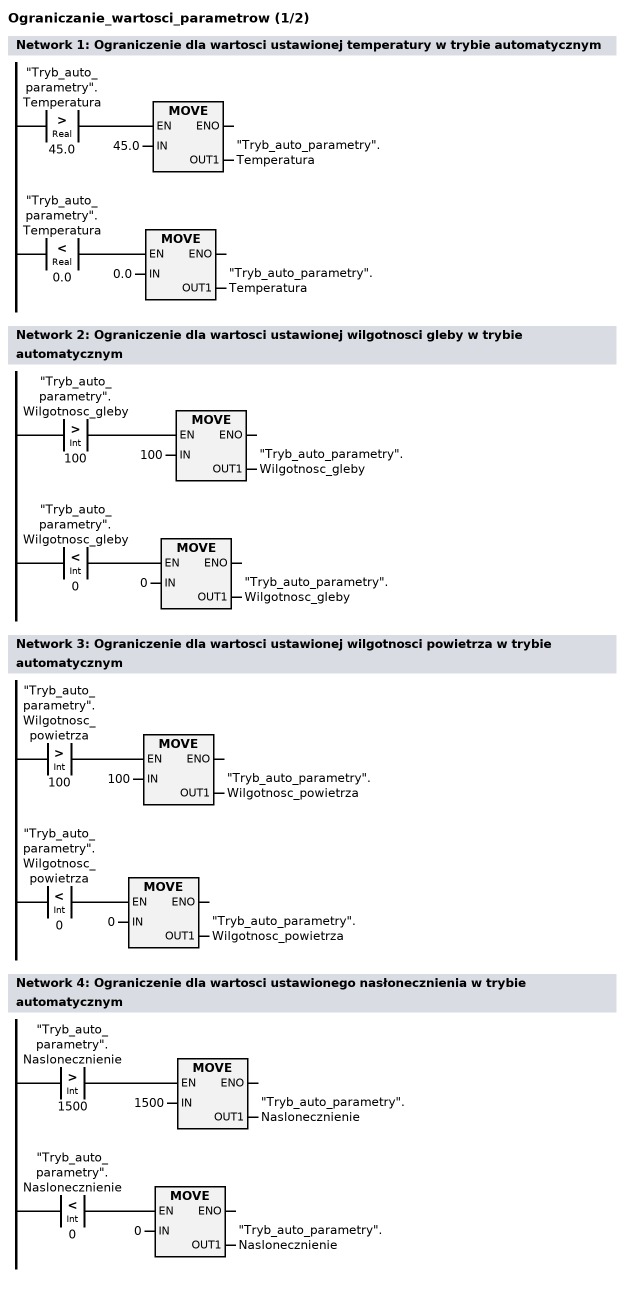
   RUNG wire#powerrail
      { S7_Templates := "SrcType := Real" } GT_Contact(in1 := "Tryb_auto_parametry".Temperatura, in2 := 45.0)
      Move(in := 45.0, out1 => "Tryb_auto_parametry".Temperatura)
   END_RUNG
   RUNG wire#powerrail
      { S7_Templates := "SrcType := Real" } LT_Contact(in1 := "Tryb_auto_parametry".Temperatura, in2 := 0.0)
      Move(in := 0.0, out1 => "Tryb_auto_parametry".Temperatura)
   END_RUNG
   // the same network as SCL:
   IF "Tryb_auto_parametry".Temperatura > 45.0 THEN "Tryb_auto_parametry".Temperatura := 45.0; END_IF;
   IF "Tryb_auto_parametry".Temperatura < 0.0 THEN "Tryb_auto_parametry".Temperatura := 0.0; END_IF;
END_REGION

REGION Network 2: Ograniczenie dla wartosci ustawionej wilgotnosci gleby w trybie automatycznym
   RUNG wire#powerrail
      { S7_Templates := "SrcType := Int" } GT_Contact(in1 := "Tryb_auto_parametry".Wilgotnosc_gleby, in2 := 100)
      Move(in := 100, out1 => "Tryb_auto_parametry".Wilgotnosc_gleby)
   END_RUNG
   RUNG wire#powerrail
      { S7_Templates := "SrcType := Int" } LT_Contact(in1 := "Tryb_auto_parametry".Wilgotnosc_gleby, in2 := 0)
      Move(in := 0, out1 => "Tryb_auto_parametry".Wilgotnosc_gleby)
   END_RUNG
   // the same network as SCL:
   IF "Tryb_auto_parametry".Wilgotnosc_gleby > 100 THEN
       "Tryb_auto_parametry".Wilgotnosc_gleby := 100;
   END_IF;
   IF "Tryb_auto_parametry".Wilgotnosc_gleby < 0 THEN "Tryb_auto_parametry".Wilgotnosc_gleby := 0; END_IF;
END_REGION

REGION Network 3: Ograniczenie dla wartosci ustawionej wilgotnosci powietrza w trybie automatycznym
   RUNG wire#powerrail
      { S7_Templates := "SrcType := Int" } GT_Contact(in1 := "Tryb_auto_parametry".Wilgotnosc_powietrza, in2 := 100)
      Move(in := 100, out1 => "Tryb_auto_parametry".Wilgotnosc_powietrza)
   END_RUNG
   RUNG wire#powerrail
      { S7_Templates := "SrcType := Int" } LT_Contact(in1 := "Tryb_auto_parametry".Wilgotnosc_powietrza, in2 := 0)
      Move(in := 0, out1 => "Tryb_auto_parametry".Wilgotnosc_powietrza)
   END_RUNG
   // the same network as SCL:
   IF "Tryb_auto_parametry".Wilgotnosc_powietrza > 100 THEN
       "Tryb_auto_parametry".Wilgotnosc_powietrza := 100;
   END_IF;
   IF "Tryb_auto_parametry".Wilgotnosc_powietrza < 0 THEN
       "Tryb_auto_parametry".Wilgotnosc_powietrza := 0;
   END_IF;
END_REGION

REGION Network 4: Ograniczenie dla wartosci ustawionego nasłonecznienia w trybie automatycznym
   RUNG wire#powerrail
      { S7_Templates := "SrcType := Int" } GT_Contact(in1 := "Tryb_auto_parametry".Naslonecznienie, in2 := 1500)
      Move(in := 1500, out1 => "Tryb_auto_parametry".Naslonecznienie)
   END_RUNG
   RUNG wire#powerrail
      { S7_Templates := "SrcType := Int" } LT_Contact(in1 := "Tryb_auto_parametry".Naslonecznienie, in2 := 0)
      Move(in := 0, out1 => "Tryb_auto_parametry".Naslonecznienie)
   END_RUNG
   // the same network as SCL:
   IF "Tryb_auto_parametry".Naslonecznienie > 1500 THEN
       "Tryb_auto_parametry".Naslonecznienie := 1500;
   END_IF;
   IF "Tryb_auto_parametry".Naslonecznienie < 0 THEN "Tryb_auto_parametry".Naslonecznienie := 0; END_IF;
END_REGION

REGION Network 5: Ograniczenie dla wartosci ustawionego stężenia CO2 w trybie automatycznym
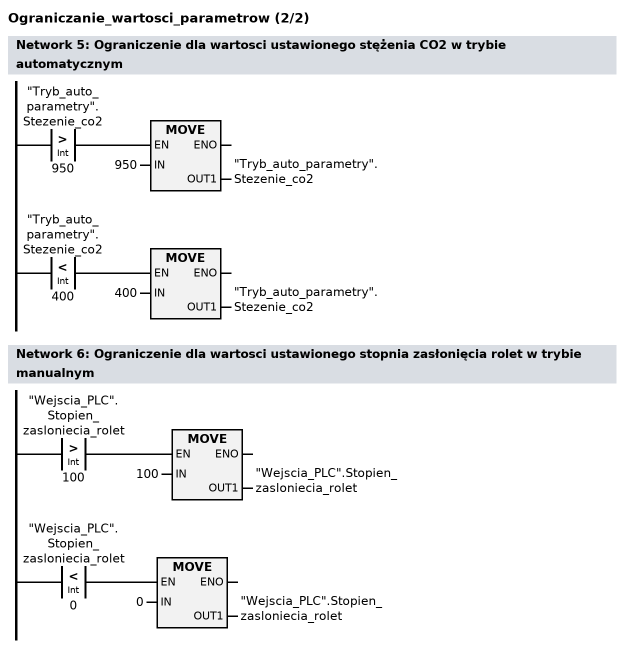
   RUNG wire#powerrail
      { S7_Templates := "SrcType := Int" } GT_Contact(in1 := "Tryb_auto_parametry".Stezenie_co2, in2 := 950)
      Move(in := 950, out1 => "Tryb_auto_parametry".Stezenie_co2)
   END_RUNG
   RUNG wire#powerrail
      { S7_Templates := "SrcType := Int" } LT_Contact(in1 := "Tryb_auto_parametry".Stezenie_co2, in2 := 400)
      Move(in := 400, out1 => "Tryb_auto_parametry".Stezenie_co2)
   END_RUNG
   // the same network as SCL:
   IF "Tryb_auto_parametry".Stezenie_co2 > 950 THEN "Tryb_auto_parametry".Stezenie_co2 := 950; END_IF;
   IF "Tryb_auto_parametry".Stezenie_co2 < 400 THEN "Tryb_auto_parametry".Stezenie_co2 := 400; END_IF;
END_REGION

REGION Network 6: Ograniczenie dla wartosci ustawionego stopnia zasłonięcia rolet w trybie manualnym
   RUNG wire#powerrail
      { S7_Templates := "SrcType := Int" } GT_Contact(in1 := "Wejscia_PLC".Stopien_zasloniecia_rolet, in2 := 100)
      Move(in := 100, out1 => "Wejscia_PLC".Stopien_zasloniecia_rolet)
   END_RUNG
   RUNG wire#powerrail
      { S7_Templates := "SrcType := Int" } LT_Contact(in1 := "Wejscia_PLC".Stopien_zasloniecia_rolet, in2 := 0)
      Move(in := 0, out1 => "Wejscia_PLC".Stopien_zasloniecia_rolet)
   END_RUNG
   // the same network as SCL:
   IF "Wejscia_PLC".Stopien_zasloniecia_rolet > 100 THEN
       "Wejscia_PLC".Stopien_zasloniecia_rolet := 100;
   END_IF;
   IF "Wejscia_PLC".Stopien_zasloniecia_rolet < 0 THEN "Wejscia_PLC".Stopien_zasloniecia_rolet := 0; END_IF;
END_REGION
END_FUNCTION

FUNCTION "Sterowanie_podlewaniem_zraszaniem" : Void   // FC7, LAD
{ S7_Optimized_Access := 'TRUE' }
VERSION : 0.1
   VAR_INPUT
      Czy_automatyczny : Bool;
      Czy_manualny : Bool;
   END_VAR
BEGIN

REGION Network 1: Sterowanie pompą zraszaczy, które odpowiadają za wilgotność powietrza w szklarni
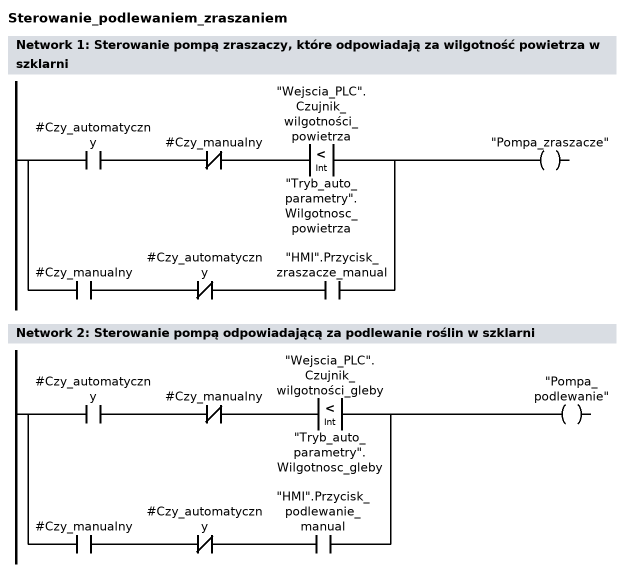
   RUNG wire#powerrail
      Contact( #Czy_automatyczny )
      I_Contact( #Czy_manualny )
      { S7_Templates := "SrcType := Int" } LT_Contact(in1 := "Wejscia_PLC".Czujnik_wilgotności_powietrza, in2 := "Tryb_auto_parametry".Wilgotnosc_powietrza)
      wire#w1
      Coil( "Pompa_zraszacze" )
   END_RUNG
   RUNG wire#powerrail
      Contact( #Czy_manualny )
      I_Contact( #Czy_automatyczny )
      Contact( "HMI".Przycisk_zraszacze_manual )
   END_RUNG wire#w1
   // the same network as SCL:
   "Pompa_zraszacze" := (#Czy_automatyczny AND NOT #Czy_manualny AND ("Wejscia_PLC".Czujnik_wilgotności_powietrza < "Tryb_auto_parametry".Wilgotnosc_powietrza)) OR (#Czy_manualny AND NOT #Czy_automatyczny AND "HMI".Przycisk_zraszacze_manual);
END_REGION

REGION Network 2: Sterowanie pompą odpowiadającą za podlewanie roślin w szklarni
   RUNG wire#powerrail
      Contact( #Czy_automatyczny )
      I_Contact( #Czy_manualny )
      { S7_Templates := "SrcType := Int" } LT_Contact(in1 := "Wejscia_PLC".Czujnik_wilgotności_gleby, in2 := "Tryb_auto_parametry".Wilgotnosc_gleby)
      wire#w1
      Coil( "Pompa_podlewanie" )
   END_RUNG
   RUNG wire#powerrail
      Contact( #Czy_manualny )
      I_Contact( #Czy_automatyczny )
      Contact( "HMI".Przycisk_podlewanie_manual )
   END_RUNG wire#w1
   // the same network as SCL:
   "Pompa_podlewanie" := (#Czy_automatyczny AND NOT #Czy_manualny AND ("Wejscia_PLC".Czujnik_wilgotności_gleby < "Tryb_auto_parametry".Wilgotnosc_gleby)) OR (#Czy_manualny AND NOT #Czy_automatyczny AND "HMI".Przycisk_podlewanie_manual);
END_REGION
END_FUNCTION

FUNCTION "Sterowanie_oknami" : Void   // FC8, LAD
{ S7_Optimized_Access := 'TRUE' }
VERSION : 0.1
   VAR_INPUT
      czy_manualny : Bool;
      czy_automatyczny : Bool;
   END_VAR
   VAR_TEMP
      Histereza_plus : Int;
      Histereza_minus : Int;
      Zakres_temp_gora : Real;   // Górny zakres temperatury zewnętrznej dla której w trybie automatycznym będą otwierane okna
      Zakres_temp_dol : Real;   // Dolny zakres temperatury zewnętrznej dla której w trybie automatycznym będą otwierane okna
   END_VAR
   VAR CONSTANT
      Histereza : Int := 25;   // Histereza, która określa kiedy stan CO2 w szklarni jest uznawany za prawidłowy
   END_VAR
BEGIN

REGION Network 1: Operacje matematyczne używane w networku 2. i 3.
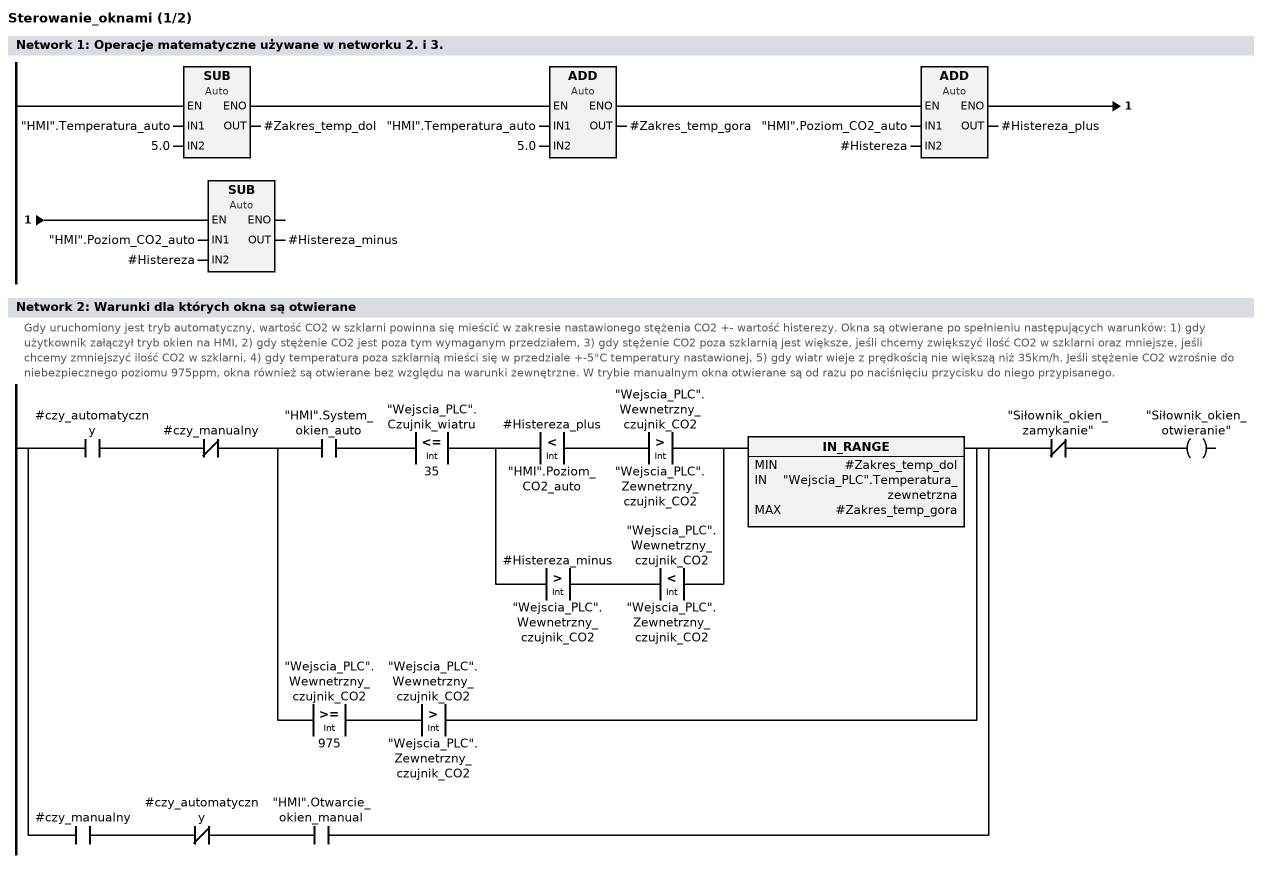
   RUNG wire#powerrail
      Sub(in1 := "HMI".Temperatura_auto, in2 := 5.0, out => #Zakres_temp_dol)
      Add(in1 := "HMI".Temperatura_auto, in2 := 5.0, out => #Zakres_temp_gora)
      Add(in1 := "HMI".Poziom_CO2_auto, in2 := #Histereza, out => #Histereza_plus)
      Sub(in1 := "HMI".Poziom_CO2_auto, in2 := #Histereza, out => #Histereza_minus)
   END_RUNG
   // the same network as SCL:
   #Zakres_temp_dol := "HMI".Temperatura_auto - 5.0;
   #Zakres_temp_gora := "HMI".Temperatura_auto + 5.0;
   #Histereza_plus := "HMI".Poziom_CO2_auto + #Histereza;
   #Histereza_minus := "HMI".Poziom_CO2_auto - #Histereza;
END_REGION

REGION Network 2: Warunki dla których okna są otwierane
   // Gdy uruchomiony jest tryb automatyczny, wartość CO2 w szklarni powinna się mieścić w zakresie nastawionego stężenia CO2 +- wartość histerezy. Okna są otwierane po spełnieniu następujących warunków: 1) gdy użytkownik załączył tryb okien na HMI, 2) gdy stężenie CO2 jest poza tym wymaganym przedziałem, 3) gdy stężenie CO2 poza szklarnią jest większe, jeśli chcemy zwiększyć ilość CO2 w szklarni oraz mniejsze, jeśli chcemy zmniejszyć ilość CO2 w szklarni, 4) gdy temperatura poza szklarnią mieści się w przedziale +-5°C temperatury nastawionej, 5) gdy wiatr wieje z prędkością nie większą niż 35km/h. Jeśli stężenie CO2 wzrośnie do niebezpiecznego poziomu 975ppm, okna również są otwierane bez względu na warunki zewnętrzne. W trybie manualnym okna otwierane są od razu po naciśnięciu przycisku do niego przypisanego.
   RUNG wire#powerrail
      Contact( #czy_automatyczny )
      I_Contact( #czy_manualny )
      wire#w1
      Contact( "HMI".System_okien_auto )
      { S7_Templates := "SrcType := Int" } LE_Contact(in1 := "Wejscia_PLC".Czujnik_wiatru, in2 := 35)
      wire#w2
      { S7_Templates := "SrcType := Int" } LT_Contact(in1 := #Histereza_plus, in2 := "HMI".Poziom_CO2_auto)
      { S7_Templates := "SrcType := Int" } GT_Contact(in1 := "Wejscia_PLC".Wewnetrzny_czujnik_CO2, in2 := "Wejscia_PLC".Zewnetrzny_czujnik_CO2)
      wire#w3
      { S7_Templates := "SrcType := Real" } InRange(min := #Zakres_temp_dol, in := "Wejscia_PLC".Temperatura_zewnetrzna, max := #Zakres_temp_gora)
      wire#w4
      I_Contact( "Siłownik_okien_zamykanie" )
      Coil( "Siłownik_okien_otwieranie" )
   END_RUNG
   RUNG wire#w2
      { S7_Templates := "SrcType := Int" } GT_Contact(in1 := #Histereza_minus, in2 := "Wejscia_PLC".Wewnetrzny_czujnik_CO2)
      { S7_Templates := "SrcType := Int" } LT_Contact(in1 := "Wejscia_PLC".Wewnetrzny_czujnik_CO2, in2 := "Wejscia_PLC".Zewnetrzny_czujnik_CO2)
   END_RUNG wire#w3
   RUNG wire#w1
      { S7_Templates := "SrcType := Int" } GE_Contact(in1 := "Wejscia_PLC".Wewnetrzny_czujnik_CO2, in2 := 975)
      { S7_Templates := "SrcType := Int" } GT_Contact(in1 := "Wejscia_PLC".Wewnetrzny_czujnik_CO2, in2 := "Wejscia_PLC".Zewnetrzny_czujnik_CO2)
   END_RUNG wire#w4
   RUNG wire#powerrail
      Contact( #czy_manualny )
      I_Contact( #czy_automatyczny )
      Contact( "HMI".Otwarcie_okien_manual )
   END_RUNG wire#w4
   // the same network as SCL:
   "Siłownik_okien_otwieranie" := ((#czy_automatyczny AND NOT #czy_manualny AND (("HMI".System_okien_auto AND ("Wejscia_PLC".Czujnik_wiatru <= 35) AND (((#Histereza_plus < "HMI".Poziom_CO2_auto) AND ("Wejscia_PLC".Wewnetrzny_czujnik_CO2 > "Wejscia_PLC".Zewnetrzny_czujnik_CO2)) OR ((#Histereza_minus > "Wejscia_PLC".Wewnetrzny_czujnik_CO2) AND ("Wejscia_PLC".Wewnetrzny_czujnik_CO2 < "Wejscia_PLC".Zewnetrzny_czujnik_CO2))) AND (#Zakres_temp_dol <= "Wejscia_PLC".Temperatura_zewnetrzna) AND ("Wejscia_PLC".Temperatura_zewnetrzna <= #Zakres_temp_gora)) OR (("Wejscia_PLC".Wewnetrzny_czujnik_CO2 >= 975) AND ("Wejscia_PLC".Wewnetrzny_czujnik_CO2 > "Wejscia_PLC".Zewnetrzny_czujnik_CO2)))) OR (#czy_manualny AND NOT #czy_automatyczny AND "HMI".Otwarcie_okien_manual)) AND NOT "Siłownik_okien_zamykanie";
END_REGION

REGION Network 3: Warunki dla których okna są zamykane
   // W trybie automatycznym okna są zamykane: 1) gdy tryb okien został wyłączony przez użytkownika, 2) gdy stężenie CO2 w szklarni wynosi zadaną wartość tego parametru +- histereza, 3) gdy stężenie CO2 poza szklarnią jest mniejsze, niż wewnątrz, jeśli chcemy zwiększyć jego ilość oraz większe, gdy chcemy zmniejszyć jego ilość, 4) gdy tempperatura zewnętrzna różni się o ponad 5°C od zadanej, 5) gdy wiatr wieje z prędkością większą niż 35km/h, 6) gdy stężenie CO2 w szklarni nie przekracza 955ppm lub przekracza, ale stężenie CO2 poza szklarnią jest większe. W trybie manualnym okna są zamykane, gdy przełączk na HMI znajdzie się w pozycji "ZAMKNIĘTE".
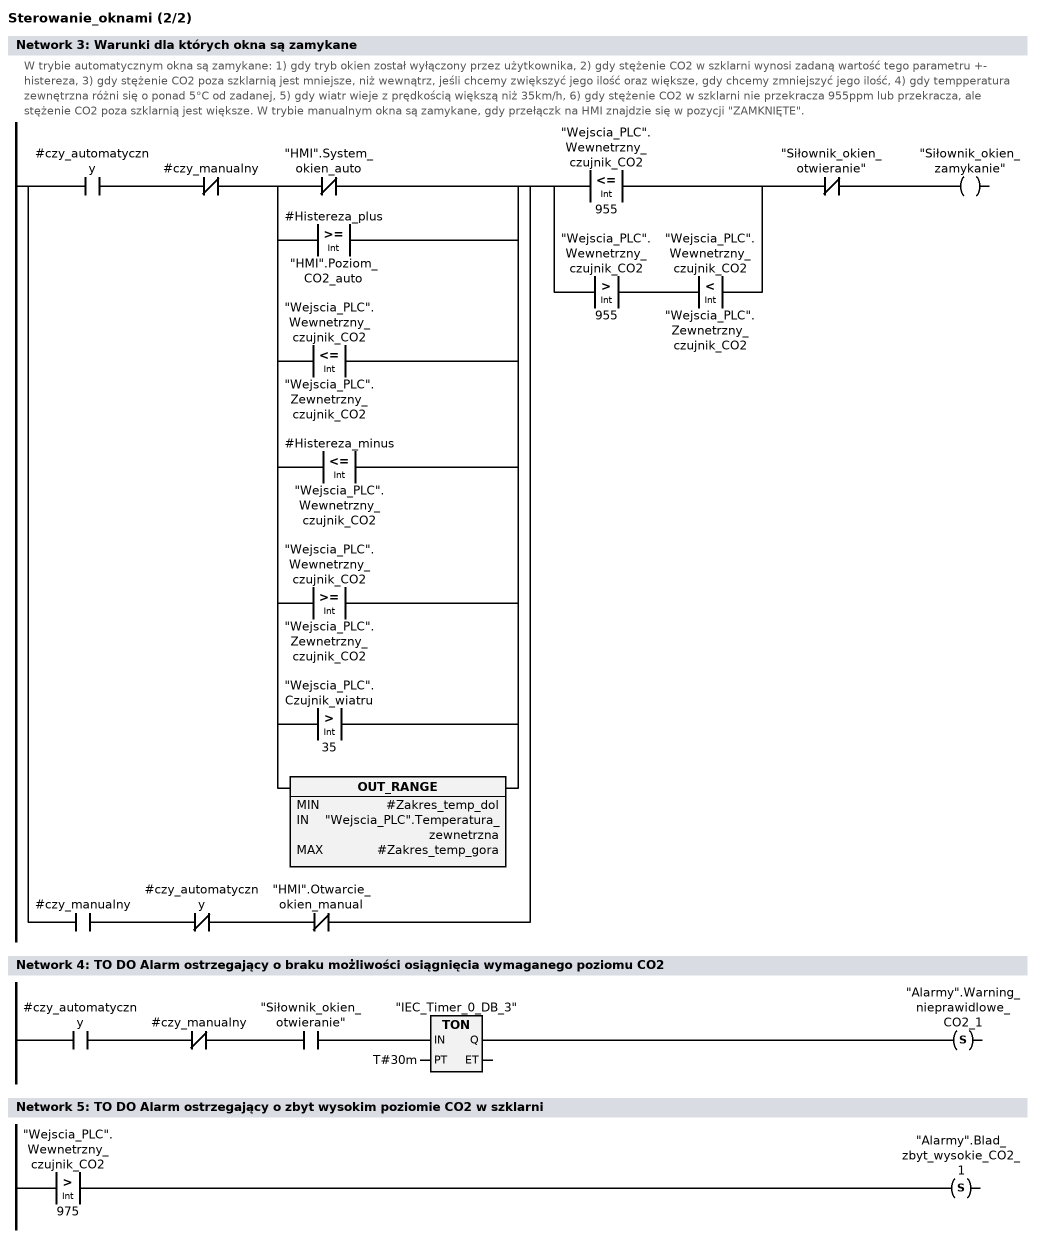
   "Siłownik_okien_zamykanie" := ((#czy_automatyczny AND NOT #czy_manualny AND (NOT "HMI".System_okien_auto OR (#Histereza_plus >= "HMI".Poziom_CO2_auto) OR ("Wejscia_PLC".Wewnetrzny_czujnik_CO2 <= "Wejscia_PLC".Zewnetrzny_czujnik_CO2) OR (#Histereza_minus <= "Wejscia_PLC".Wewnetrzny_czujnik_CO2) OR ("Wejscia_PLC".Wewnetrzny_czujnik_CO2 >= "Wejscia_PLC".Zewnetrzny_czujnik_CO2) OR ("Wejscia_PLC".Czujnik_wiatru > 35) OR ("Wejscia_PLC".Temperatura_zewnetrzna < #Zakres_temp_dol) OR ("Wejscia_PLC".Temperatura_zewnetrzna > #Zakres_temp_gora))) OR (#czy_manualny AND NOT #czy_automatyczny AND NOT "HMI".Otwarcie_okien_manual)) AND (("Wejscia_PLC".Wewnetrzny_czujnik_CO2 <= 955) OR (("Wejscia_PLC".Wewnetrzny_czujnik_CO2 > 955) AND ("Wejscia_PLC".Wewnetrzny_czujnik_CO2 < "Wejscia_PLC".Zewnetrzny_czujnik_CO2))) AND NOT "Siłownik_okien_otwieranie";
END_REGION

REGION Network 4: TO DO Alarm ostrzegający o braku możliwości osiągnięcia wymaganego poziomu CO2
   "IEC_Timer_0_DB_3".TON(IN := #czy_automatyczny AND NOT #czy_manualny AND "Siłownik_okien_otwieranie",
                          PT := T#30m);
   IF "IEC_Timer_0_DB_3".Q THEN "Alarmy".Warning_nieprawidlowe_CO2_1 := TRUE; END_IF;
END_REGION

REGION Network 5: TO DO Alarm ostrzegający o zbyt wysokim poziomie CO2 w szklarni
   RUNG wire#powerrail
      { S7_Templates := "SrcType := Int" } GT_Contact(in1 := "Wejscia_PLC".Wewnetrzny_czujnik_CO2, in2 := 975)
      S_Coil( "Alarmy".Blad_zbyt_wysokie_CO2_1 )
   END_RUNG
   // the same network as SCL:
   IF "Wejscia_PLC".Wewnetrzny_czujnik_CO2 > 975 THEN "Alarmy".Blad_zbyt_wysokie_CO2_1 := TRUE; END_IF;
END_REGION
END_FUNCTION

FUNCTION "SYMULACJA" : Void   // FC9, LAD
{ S7_Optimized_Access := 'TRUE' }
VERSION : 0.1
   VAR_INPUT
      counters : Bool;
   END_VAR
   VAR_TEMP
      temperatura_temp : Real;
      roznica_temperatur : Real;
      "wilgotność powietrza_temp" : Int;
      wilgotnosc_gleby_temp : Int;
      stezenie_CO2 : Int;
      natezenie_swiatla_temp : Int;
      odsloniecie_okna_temp : Real;
      pedkosc_wiatru_temp : Real;
      rand : Real;
      error : Bool;
      status : Int;
      sub_status : Int;
      rolety_temp : Real;
   END_VAR
   VAR_TEMP   // added for the SCL form of the ladder/FBD networks
      _w1 : Bool;
   END_VAR
BEGIN

REGION Network 1: blok oblicza roznice temperatur
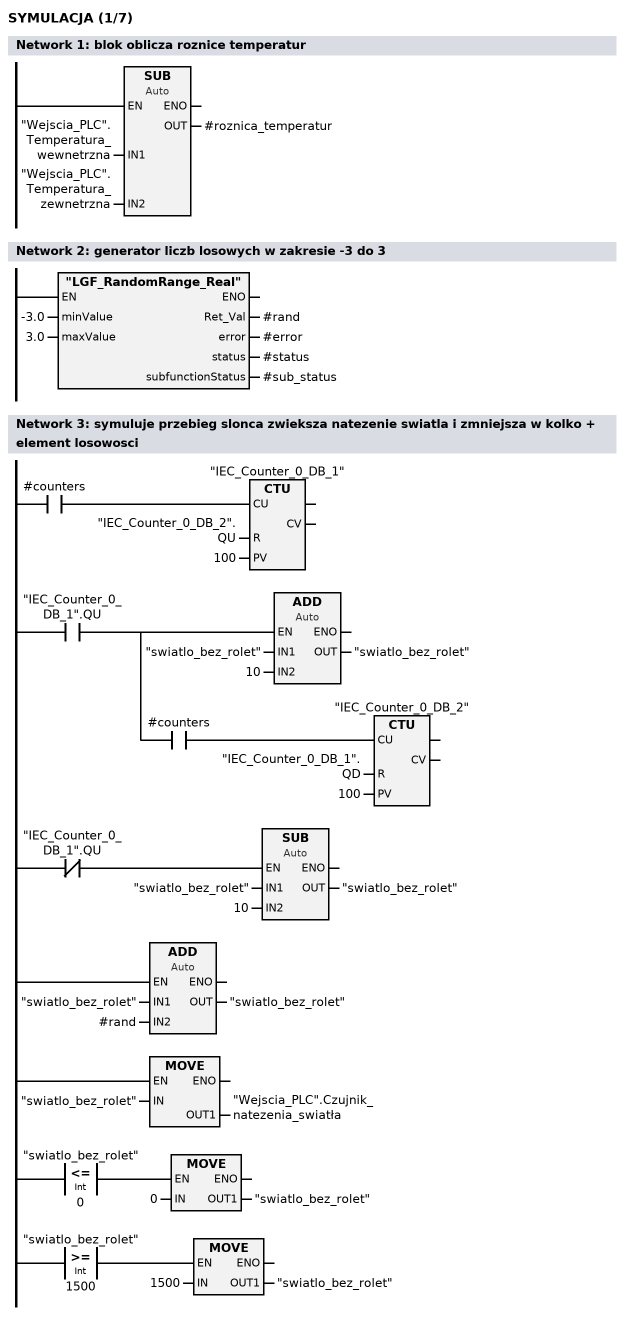
   RUNG wire#powerrail
      Sub(in1 := "Wejscia_PLC".Temperatura_wewnetrzna, in2 := "Wejscia_PLC".Temperatura_zewnetrzna, out => #roznica_temperatur)
   END_RUNG
   // the same network as SCL:
   #roznica_temperatur := "Wejscia_PLC".Temperatura_wewnetrzna - "Wejscia_PLC".Temperatura_zewnetrzna;
END_REGION

REGION Network 2: generator liczb losowych w zakresie -3 do 3
   RUNG wire#powerrail
      "LGF_RandomRange_Real"(minValue := -3.0, maxValue := 3.0, Ret_Val => #rand, error => #error, status => #status, subfunctionStatus => #sub_status)
   END_RUNG
   // the same network as SCL:
   #rand := "LGF_RandomRange_Real"(minValue := -3.0,
                           maxValue := 3.0,
                           error => #error,
                           status => #status,
                           subfunctionStatus => #sub_status);
END_REGION

REGION Network 3: symuluje przebieg slonca zwieksza natezenie swiatla i zmniejsza w kolko + element losowosci
   "IEC_Counter_0_DB_1".CTU(CU := #counters, R := "IEC_Counter_0_DB_2".QU, PV := 100);
   IF "IEC_Counter_0_DB_1".QU THEN "swiatlo_bez_rolet" := "swiatlo_bez_rolet" + 10; END_IF;
   "IEC_Counter_0_DB_2".CTU(CU := "IEC_Counter_0_DB_1".QU AND #counters,
                           R := "IEC_Counter_0_DB_1".QD,
                           PV := 100);
   IF NOT "IEC_Counter_0_DB_1".QU THEN "swiatlo_bez_rolet" := "swiatlo_bez_rolet" - 10; END_IF;
   "swiatlo_bez_rolet" := "swiatlo_bez_rolet" + #rand;
   "Wejscia_PLC".Czujnik_natezenia_swiatła := "swiatlo_bez_rolet";
   IF "swiatlo_bez_rolet" <= 0 THEN "swiatlo_bez_rolet" := 0; END_IF;
   IF "swiatlo_bez_rolet" >= 1500 THEN "swiatlo_bez_rolet" := 1500; END_IF;
END_REGION

REGION Network 4: funkcja oblicza liniową zależność natężenia światła od zasłonięcia rolet
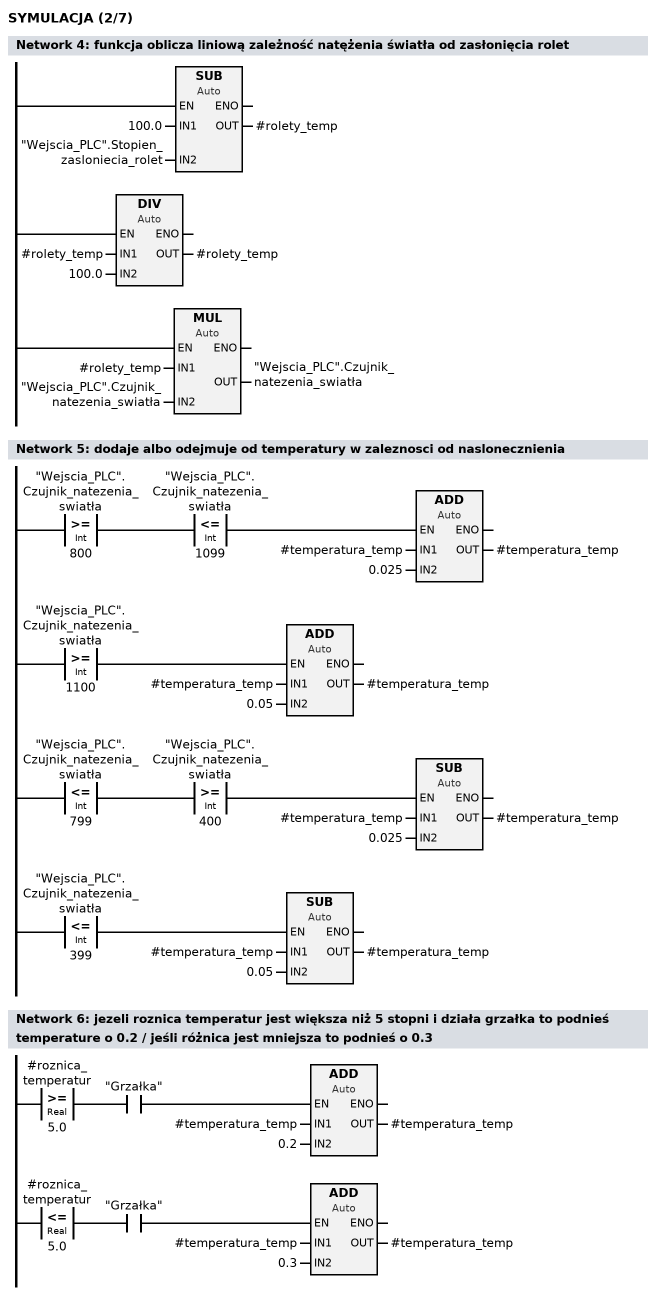
   RUNG wire#powerrail
      Sub(in1 := 100.0, in2 := "Wejscia_PLC".Stopien_zasloniecia_rolet, out => #rolety_temp)
   END_RUNG
   RUNG wire#powerrail
      Div(in1 := #rolety_temp, in2 := 100.0, out => #rolety_temp)
   END_RUNG
   RUNG wire#powerrail
      Mul(in1 := #rolety_temp, in2 := "Wejscia_PLC".Czujnik_natezenia_swiatła, out => "Wejscia_PLC".Czujnik_natezenia_swiatła)
   END_RUNG
   // the same network as SCL:
   #rolety_temp := 100.0 - "Wejscia_PLC".Stopien_zasloniecia_rolet;
   #rolety_temp := #rolety_temp / 100.0;
   "Wejscia_PLC".Czujnik_natezenia_swiatła := #rolety_temp * "Wejscia_PLC".Czujnik_natezenia_swiatła;
END_REGION

REGION Network 5: dodaje albo odejmuje od temperatury w zaleznosci od naslonecznienia
   RUNG wire#powerrail
      { S7_Templates := "SrcType := Int" } GE_Contact(in1 := "Wejscia_PLC".Czujnik_natezenia_swiatła, in2 := 800)
      { S7_Templates := "SrcType := Int" } LE_Contact(in1 := "Wejscia_PLC".Czujnik_natezenia_swiatła, in2 := 1099)
      Add(in1 := #temperatura_temp, in2 := 0.025, out => #temperatura_temp)
   END_RUNG
   RUNG wire#powerrail
      { S7_Templates := "SrcType := Int" } GE_Contact(in1 := "Wejscia_PLC".Czujnik_natezenia_swiatła, in2 := 1100)
      Add(in1 := #temperatura_temp, in2 := 0.05, out => #temperatura_temp)
   END_RUNG
   RUNG wire#powerrail
      { S7_Templates := "SrcType := Int" } LE_Contact(in1 := "Wejscia_PLC".Czujnik_natezenia_swiatła, in2 := 799)
      { S7_Templates := "SrcType := Int" } GE_Contact(in1 := "Wejscia_PLC".Czujnik_natezenia_swiatła, in2 := 400)
      Sub(in1 := #temperatura_temp, in2 := 0.025, out => #temperatura_temp)
   END_RUNG
   RUNG wire#powerrail
      { S7_Templates := "SrcType := Int" } LE_Contact(in1 := "Wejscia_PLC".Czujnik_natezenia_swiatła, in2 := 399)
      Sub(in1 := #temperatura_temp, in2 := 0.05, out => #temperatura_temp)
   END_RUNG
   // the same network as SCL:
   IF ("Wejscia_PLC".Czujnik_natezenia_swiatła >= 800) AND ("Wejscia_PLC".Czujnik_natezenia_swiatła <= 1099) THEN
       #temperatura_temp := #temperatura_temp + 0.025;
   END_IF;
   IF "Wejscia_PLC".Czujnik_natezenia_swiatła >= 1100 THEN
       #temperatura_temp := #temperatura_temp + 0.05;
   END_IF;
   IF ("Wejscia_PLC".Czujnik_natezenia_swiatła <= 799) AND ("Wejscia_PLC".Czujnik_natezenia_swiatła >= 400) THEN
       #temperatura_temp := #temperatura_temp - 0.025;
   END_IF;
   IF "Wejscia_PLC".Czujnik_natezenia_swiatła <= 399 THEN
       #temperatura_temp := #temperatura_temp - 0.05;
   END_IF;
END_REGION

REGION Network 6: jezeli roznica temperatur jest większa niż 5 stopni i działa grzałka to podnieś temperature o 0.2 / jeśli różnica jest mniejsza to podnieś o 0.3
   RUNG wire#powerrail
      { S7_Templates := "SrcType := Real" } GE_Contact(in1 := #roznica_temperatur, in2 := 5.0)
      Contact( "Grzałka" )
      Add(in1 := #temperatura_temp, in2 := 0.2, out => #temperatura_temp)
   END_RUNG
   RUNG wire#powerrail
      { S7_Templates := "SrcType := Real" } LE_Contact(in1 := #roznica_temperatur, in2 := 5.0)
      Contact( "Grzałka" )
      Add(in1 := #temperatura_temp, in2 := 0.3, out => #temperatura_temp)
   END_RUNG
   // the same network as SCL:
   IF (#roznica_temperatur >= 5.0) AND "Grzałka" THEN #temperatura_temp := #temperatura_temp + 0.2; END_IF;
   IF (#roznica_temperatur <= 5.0) AND "Grzałka" THEN #temperatura_temp := #temperatura_temp + 0.3; END_IF;
END_REGION

REGION Network 7: jezeli działa wentylator to obniż temperature o 0.1
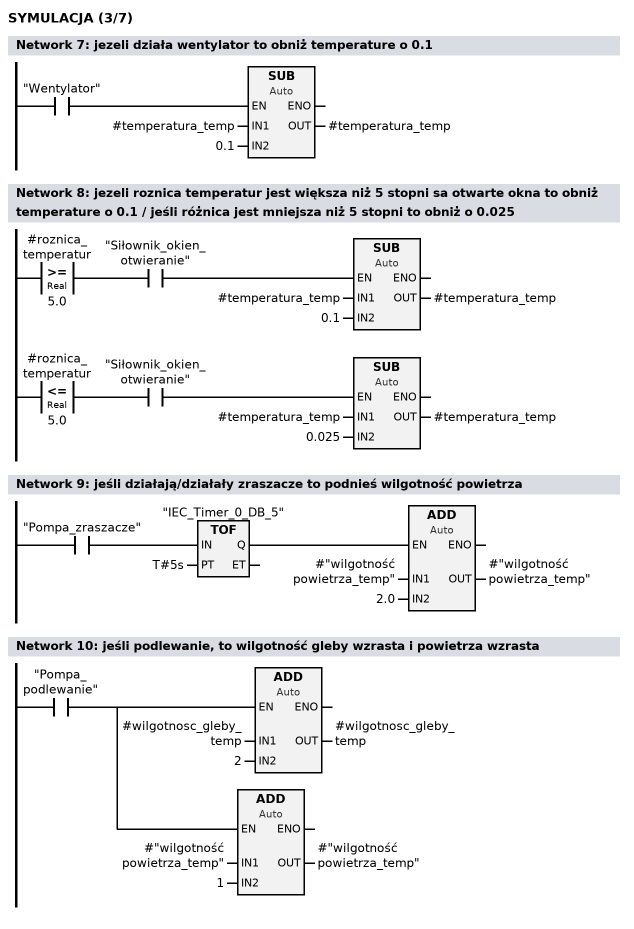
   RUNG wire#powerrail
      Contact( "Wentylator" )
      Sub(in1 := #temperatura_temp, in2 := 0.1, out => #temperatura_temp)
   END_RUNG
   // the same network as SCL:
   IF "Wentylator" THEN #temperatura_temp := #temperatura_temp - 0.1; END_IF;
END_REGION

REGION Network 8: jezeli roznica temperatur jest większa niż 5 stopni sa otwarte okna to obniż temperature o 0.1 / jeśli różnica jest mniejsza niż 5 stopni to obniż o 0.025
   RUNG wire#powerrail
      { S7_Templates := "SrcType := Real" } GE_Contact(in1 := #roznica_temperatur, in2 := 5.0)
      Contact( "Siłownik_okien_otwieranie" )
      Sub(in1 := #temperatura_temp, in2 := 0.1, out => #temperatura_temp)
   END_RUNG
   RUNG wire#powerrail
      { S7_Templates := "SrcType := Real" } LE_Contact(in1 := #roznica_temperatur, in2 := 5.0)
      Contact( "Siłownik_okien_otwieranie" )
      Sub(in1 := #temperatura_temp, in2 := 0.025, out => #temperatura_temp)
   END_RUNG
   // the same network as SCL:
   IF (#roznica_temperatur >= 5.0) AND "Siłownik_okien_otwieranie" THEN
       #temperatura_temp := #temperatura_temp - 0.1;
   END_IF;
   IF (#roznica_temperatur <= 5.0) AND "Siłownik_okien_otwieranie" THEN
       #temperatura_temp := #temperatura_temp - 0.025;
   END_IF;
END_REGION

REGION Network 9: jeśli działają/działały zraszacze to podnieś wilgotność powietrza
   "IEC_Timer_0_DB_5".TOF(IN := "Pompa_zraszacze", PT := T#5s);
   IF "IEC_Timer_0_DB_5".Q THEN #"wilgotność powietrza_temp" := #"wilgotność powietrza_temp" + 2.0; END_IF;
END_REGION

REGION Network 10: jeśli podlewanie, to wilgotność gleby wzrasta i powietrza wzrasta
   RUNG wire#powerrail
      Contact( "Pompa_podlewanie" )
      wire#w1
      Add(in1 := #wilgotnosc_gleby_temp, in2 := 2, out => #wilgotnosc_gleby_temp)
   END_RUNG
   RUNG wire#w1
      Add(in1 := #"wilgotność powietrza_temp", in2 := 1, out => #"wilgotność powietrza_temp")
   END_RUNG
   // the same network as SCL:
   IF "Pompa_podlewanie" THEN
       #wilgotnosc_gleby_temp := #wilgotnosc_gleby_temp + 2;
       #"wilgotność powietrza_temp" := #"wilgotność powietrza_temp" + 1;
   END_IF;
END_REGION

REGION Network 11: realizacja zaleznosci odslaniania i zaslaniania rolet, od stopnia zasłonięcia
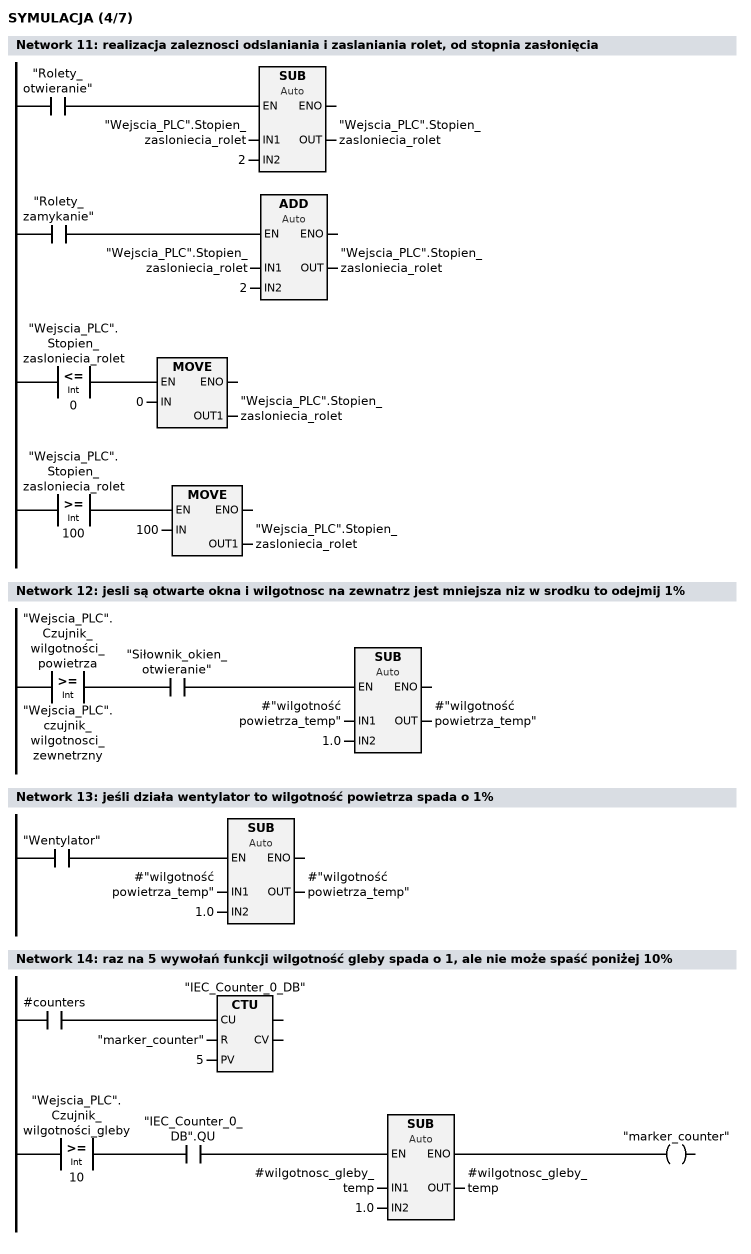
   RUNG wire#powerrail
      Contact( "Rolety_otwieranie" )
      Sub(in1 := "Wejscia_PLC".Stopien_zasloniecia_rolet, in2 := 2, out => "Wejscia_PLC".Stopien_zasloniecia_rolet)
   END_RUNG
   RUNG wire#powerrail
      Contact( "Rolety_zamykanie" )
      Add(in1 := "Wejscia_PLC".Stopien_zasloniecia_rolet, in2 := 2, out => "Wejscia_PLC".Stopien_zasloniecia_rolet)
   END_RUNG
   RUNG wire#powerrail
      { S7_Templates := "SrcType := Int" } LE_Contact(in1 := "Wejscia_PLC".Stopien_zasloniecia_rolet, in2 := 0)
      Move(in := 0, out1 => "Wejscia_PLC".Stopien_zasloniecia_rolet)
   END_RUNG
   RUNG wire#powerrail
      { S7_Templates := "SrcType := Int" } GE_Contact(in1 := "Wejscia_PLC".Stopien_zasloniecia_rolet, in2 := 100)
      Move(in := 100, out1 => "Wejscia_PLC".Stopien_zasloniecia_rolet)
   END_RUNG
   // the same network as SCL:
   IF "Rolety_otwieranie" THEN
       "Wejscia_PLC".Stopien_zasloniecia_rolet := "Wejscia_PLC".Stopien_zasloniecia_rolet - 2;
   END_IF;
   IF "Rolety_zamykanie" THEN
       "Wejscia_PLC".Stopien_zasloniecia_rolet := "Wejscia_PLC".Stopien_zasloniecia_rolet + 2;
   END_IF;
   IF "Wejscia_PLC".Stopien_zasloniecia_rolet <= 0 THEN "Wejscia_PLC".Stopien_zasloniecia_rolet := 0; END_IF;
   IF "Wejscia_PLC".Stopien_zasloniecia_rolet >= 100 THEN
       "Wejscia_PLC".Stopien_zasloniecia_rolet := 100;
   END_IF;
END_REGION

REGION Network 12: jesli są otwarte okna i wilgotnosc na zewnatrz jest mniejsza niz w srodku to odejmij 1%
   RUNG wire#powerrail
      { S7_Templates := "SrcType := Int" } GE_Contact(in1 := "Wejscia_PLC".Czujnik_wilgotności_powietrza, in2 := "Wejscia_PLC".czujnik_wilgotnosci_zewnetrzny)
      Contact( "Siłownik_okien_otwieranie" )
      Sub(in1 := #"wilgotność powietrza_temp", in2 := 1.0, out => #"wilgotność powietrza_temp")
   END_RUNG
   // the same network as SCL:
   IF ("Wejscia_PLC".Czujnik_wilgotności_powietrza >= "Wejscia_PLC".czujnik_wilgotnosci_zewnetrzny) AND "Siłownik_okien_otwieranie" THEN
       #"wilgotność powietrza_temp" := #"wilgotność powietrza_temp" - 1.0;
   END_IF;
END_REGION

REGION Network 13: jeśli działa wentylator to wilgotność powietrza spada o 1%
   RUNG wire#powerrail
      Contact( "Wentylator" )
      Sub(in1 := #"wilgotność powietrza_temp", in2 := 1.0, out => #"wilgotność powietrza_temp")
   END_RUNG
   // the same network as SCL:
   IF "Wentylator" THEN #"wilgotność powietrza_temp" := #"wilgotność powietrza_temp" - 1.0; END_IF;
END_REGION

REGION Network 14: raz na 5 wywołań funkcji wilgotność gleby spada o 1, ale nie może spaść poniżej 10%
   "IEC_Counter_0_DB".CTU(CU := #counters, R := "marker_counter", PV := 5);
   #_w1 := ("Wejscia_PLC".Czujnik_wilgotności_gleby >= 10) AND "IEC_Counter_0_DB".QU;
   IF #_w1 THEN #wilgotnosc_gleby_temp := #wilgotnosc_gleby_temp - 1.0; END_IF;
   "marker_counter" := #_w1;
END_REGION

REGION Network 15: jeśli stężenie na zewnątrz jest mniejsze, a są otwarte okna to zmniejsz stężenie CO2
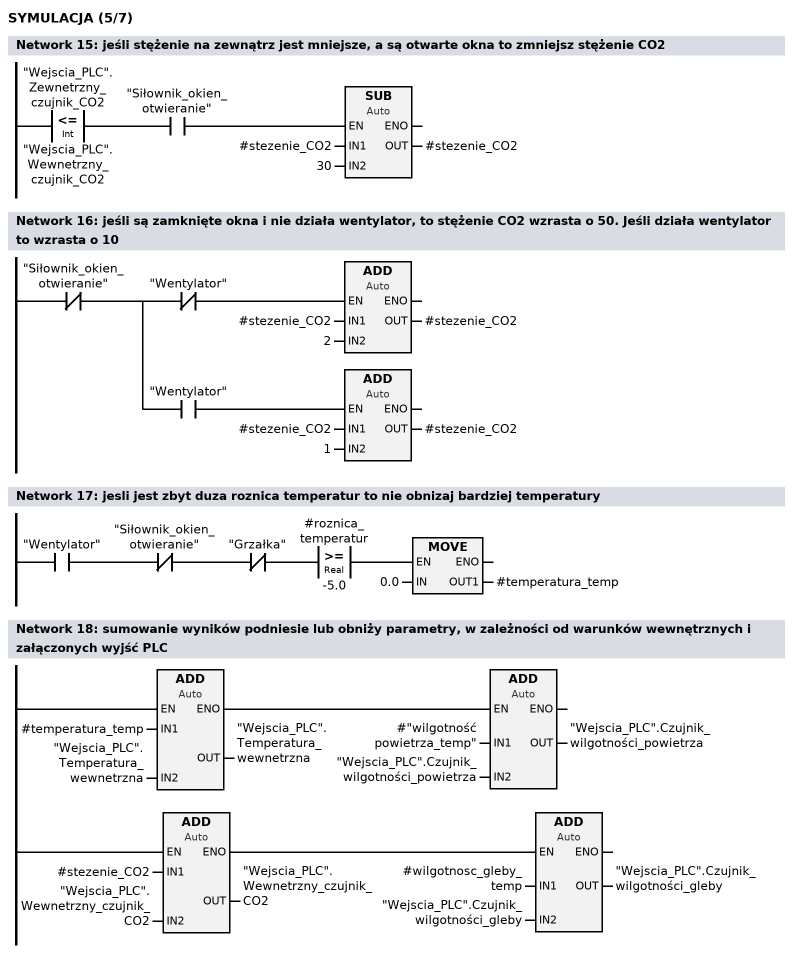
   RUNG wire#powerrail
      { S7_Templates := "SrcType := Int" } LE_Contact(in1 := "Wejscia_PLC".Zewnetrzny_czujnik_CO2, in2 := "Wejscia_PLC".Wewnetrzny_czujnik_CO2)
      Contact( "Siłownik_okien_otwieranie" )
      Sub(in1 := #stezenie_CO2, in2 := 30, out => #stezenie_CO2)
   END_RUNG
   // the same network as SCL:
   IF ("Wejscia_PLC".Zewnetrzny_czujnik_CO2 <= "Wejscia_PLC".Wewnetrzny_czujnik_CO2) AND "Siłownik_okien_otwieranie" THEN
       #stezenie_CO2 := #stezenie_CO2 - 30;
   END_IF;
END_REGION

REGION Network 16: jeśli są zamknięte okna i nie działa wentylator, to stężenie CO2 wzrasta o 50. Jeśli działa wentylator to wzrasta o 10
   RUNG wire#powerrail
      I_Contact( "Siłownik_okien_otwieranie" )
      wire#w1
      I_Contact( "Wentylator" )
      Add(in1 := #stezenie_CO2, in2 := 2, out => #stezenie_CO2)
   END_RUNG
   RUNG wire#w1
      Contact( "Wentylator" )
      Add(in1 := #stezenie_CO2, in2 := 1, out => #stezenie_CO2)
   END_RUNG
   // the same network as SCL:
   #_w1 := NOT "Siłownik_okien_otwieranie";
   IF #_w1 AND NOT "Wentylator" THEN #stezenie_CO2 := #stezenie_CO2 + 2; END_IF;
   IF #_w1 AND "Wentylator" THEN #stezenie_CO2 := #stezenie_CO2 + 1; END_IF;
END_REGION

REGION Network 17: jesli jest zbyt duza roznica temperatur to nie obnizaj bardziej temperatury
   RUNG wire#powerrail
      Contact( "Wentylator" )
      I_Contact( "Siłownik_okien_otwieranie" )
      I_Contact( "Grzałka" )
      { S7_Templates := "SrcType := Real" } GE_Contact(in1 := #roznica_temperatur, in2 := -5.0)
      Move(in := 0.0, out1 => #temperatura_temp)
   END_RUNG
   // the same network as SCL:
   IF "Wentylator" AND NOT "Siłownik_okien_otwieranie" AND NOT "Grzałka" AND (#roznica_temperatur >= (-5.0)) THEN
       #temperatura_temp := 0.0;
   END_IF;
END_REGION

REGION Network 18: sumowanie wyników podniesie lub obniży parametry, w zależności od warunków wewnętrznych i załączonych wyjść PLC
   RUNG wire#powerrail
      Add(in1 := #temperatura_temp, in2 := "Wejscia_PLC".Temperatura_wewnetrzna, out => "Wejscia_PLC".Temperatura_wewnetrzna)
      Add(in1 := #"wilgotność powietrza_temp", in2 := "Wejscia_PLC".Czujnik_wilgotności_powietrza, out => "Wejscia_PLC".Czujnik_wilgotności_powietrza)
   END_RUNG
   RUNG wire#powerrail
      Add(in1 := #stezenie_CO2, in2 := "Wejscia_PLC".Wewnetrzny_czujnik_CO2, out => "Wejscia_PLC".Wewnetrzny_czujnik_CO2)
      Add(in1 := #wilgotnosc_gleby_temp, in2 := "Wejscia_PLC".Czujnik_wilgotności_gleby, out => "Wejscia_PLC".Czujnik_wilgotności_gleby)
   END_RUNG
   // the same network as SCL:
   "Wejscia_PLC".Temperatura_wewnetrzna := #temperatura_temp + "Wejscia_PLC".Temperatura_wewnetrzna;
   "Wejscia_PLC".Czujnik_wilgotności_powietrza := #"wilgotność powietrza_temp" + "Wejscia_PLC".Czujnik_wilgotności_powietrza;
   "Wejscia_PLC".Wewnetrzny_czujnik_CO2 := #stezenie_CO2 + "Wejscia_PLC".Wewnetrzny_czujnik_CO2;
   "Wejscia_PLC".Czujnik_wilgotności_gleby := #wilgotnosc_gleby_temp + "Wejscia_PLC".Czujnik_wilgotności_gleby;
END_REGION

REGION Network 19: zabezpieczenie, przed przekroczeniem wartości krytycznych czujników + zabezpieczenia fizyczne np. procenty tylko w zakresie(0-100)
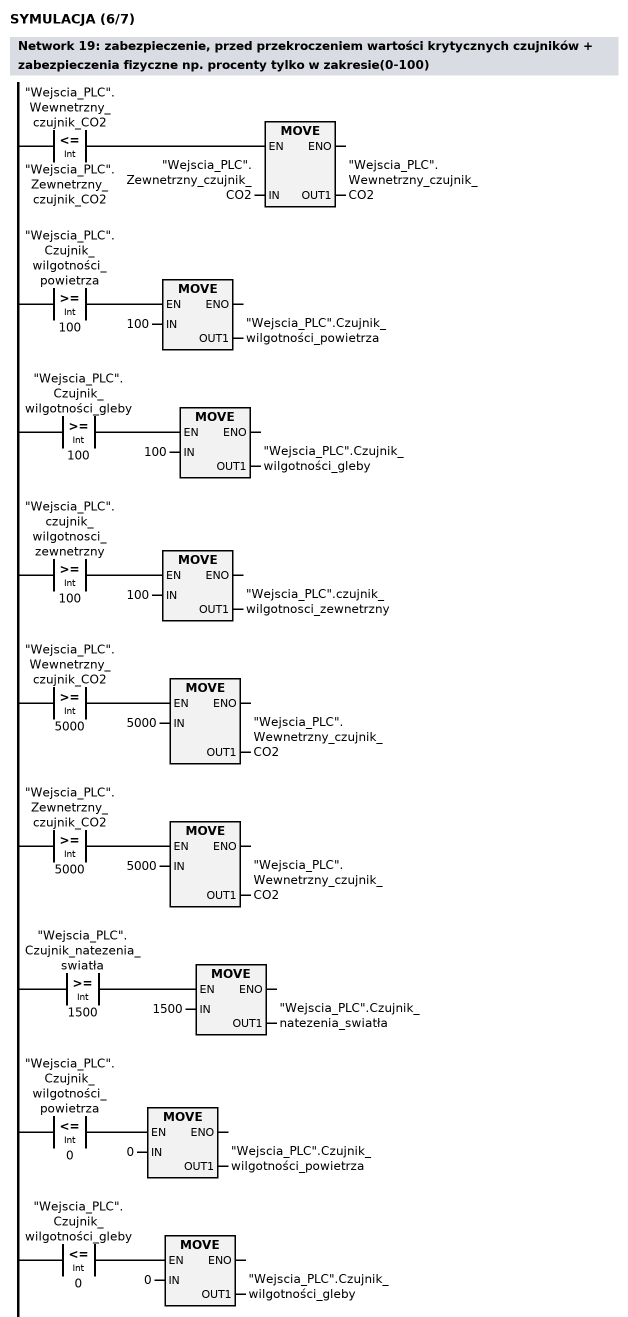
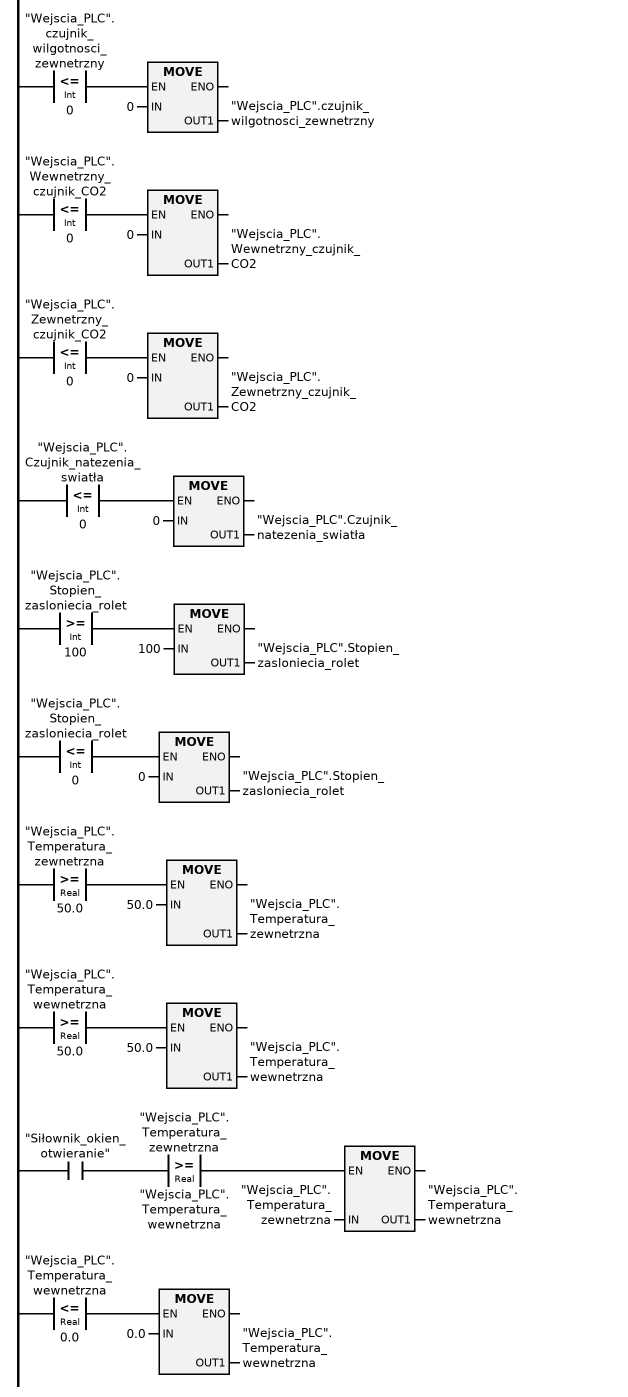
   RUNG wire#powerrail
      { S7_Templates := "SrcType := Int" } LE_Contact(in1 := "Wejscia_PLC".Wewnetrzny_czujnik_CO2, in2 := "Wejscia_PLC".Zewnetrzny_czujnik_CO2)
      Move(in := "Wejscia_PLC".Zewnetrzny_czujnik_CO2, out1 => "Wejscia_PLC".Wewnetrzny_czujnik_CO2)
   END_RUNG
   RUNG wire#powerrail
      { S7_Templates := "SrcType := Int" } GE_Contact(in1 := "Wejscia_PLC".Czujnik_wilgotności_powietrza, in2 := 100)
      Move(in := 100, out1 => "Wejscia_PLC".Czujnik_wilgotności_powietrza)
   END_RUNG
   RUNG wire#powerrail
      { S7_Templates := "SrcType := Int" } GE_Contact(in1 := "Wejscia_PLC".Czujnik_wilgotności_gleby, in2 := 100)
      Move(in := 100, out1 => "Wejscia_PLC".Czujnik_wilgotności_gleby)
   END_RUNG
   RUNG wire#powerrail
      { S7_Templates := "SrcType := Int" } GE_Contact(in1 := "Wejscia_PLC".czujnik_wilgotnosci_zewnetrzny, in2 := 100)
      Move(in := 100, out1 => "Wejscia_PLC".czujnik_wilgotnosci_zewnetrzny)
   END_RUNG
   RUNG wire#powerrail
      { S7_Templates := "SrcType := Int" } GE_Contact(in1 := "Wejscia_PLC".Wewnetrzny_czujnik_CO2, in2 := 5000)
      Move(in := 5000, out1 => "Wejscia_PLC".Wewnetrzny_czujnik_CO2)
   END_RUNG
   RUNG wire#powerrail
      { S7_Templates := "SrcType := Int" } GE_Contact(in1 := "Wejscia_PLC".Zewnetrzny_czujnik_CO2, in2 := 5000)
      Move(in := 5000, out1 => "Wejscia_PLC".Wewnetrzny_czujnik_CO2)
   END_RUNG
   RUNG wire#powerrail
      { S7_Templates := "SrcType := Int" } GE_Contact(in1 := "Wejscia_PLC".Czujnik_natezenia_swiatła, in2 := 1500)
      Move(in := 1500, out1 => "Wejscia_PLC".Czujnik_natezenia_swiatła)
   END_RUNG
   RUNG wire#powerrail
      { S7_Templates := "SrcType := Int" } LE_Contact(in1 := "Wejscia_PLC".Czujnik_wilgotności_powietrza, in2 := 0)
      Move(in := 0, out1 => "Wejscia_PLC".Czujnik_wilgotności_powietrza)
   END_RUNG
   RUNG wire#powerrail
      { S7_Templates := "SrcType := Int" } LE_Contact(in1 := "Wejscia_PLC".Czujnik_wilgotności_gleby, in2 := 0)
      Move(in := 0, out1 => "Wejscia_PLC".Czujnik_wilgotności_gleby)
   END_RUNG
   RUNG wire#powerrail
      { S7_Templates := "SrcType := Int" } LE_Contact(in1 := "Wejscia_PLC".czujnik_wilgotnosci_zewnetrzny, in2 := 0)
      Move(in := 0, out1 => "Wejscia_PLC".czujnik_wilgotnosci_zewnetrzny)
   END_RUNG
   RUNG wire#powerrail
      { S7_Templates := "SrcType := Int" } LE_Contact(in1 := "Wejscia_PLC".Wewnetrzny_czujnik_CO2, in2 := 0)
      Move(in := 0, out1 => "Wejscia_PLC".Wewnetrzny_czujnik_CO2)
   END_RUNG
   RUNG wire#powerrail
      { S7_Templates := "SrcType := Int" } LE_Contact(in1 := "Wejscia_PLC".Zewnetrzny_czujnik_CO2, in2 := 0)
      Move(in := 0, out1 => "Wejscia_PLC".Zewnetrzny_czujnik_CO2)
   END_RUNG
   RUNG wire#powerrail
      { S7_Templates := "SrcType := Int" } LE_Contact(in1 := "Wejscia_PLC".Czujnik_natezenia_swiatła, in2 := 0)
      Move(in := 0, out1 => "Wejscia_PLC".Czujnik_natezenia_swiatła)
   END_RUNG
   RUNG wire#powerrail
      { S7_Templates := "SrcType := Int" } GE_Contact(in1 := "Wejscia_PLC".Stopien_zasloniecia_rolet, in2 := 100)
      Move(in := 100, out1 => "Wejscia_PLC".Stopien_zasloniecia_rolet)
   END_RUNG
   RUNG wire#powerrail
      { S7_Templates := "SrcType := Int" } LE_Contact(in1 := "Wejscia_PLC".Stopien_zasloniecia_rolet, in2 := 0)
      Move(in := 0, out1 => "Wejscia_PLC".Stopien_zasloniecia_rolet)
   END_RUNG
   RUNG wire#powerrail
      { S7_Templates := "SrcType := Real" } GE_Contact(in1 := "Wejscia_PLC".Temperatura_zewnetrzna, in2 := 50.0)
      Move(in := 50.0, out1 => "Wejscia_PLC".Temperatura_zewnetrzna)
   END_RUNG
   RUNG wire#powerrail
      { S7_Templates := "SrcType := Real" } GE_Contact(in1 := "Wejscia_PLC".Temperatura_wewnetrzna, in2 := 50.0)
      Move(in := 50.0, out1 => "Wejscia_PLC".Temperatura_wewnetrzna)
   END_RUNG
   RUNG wire#powerrail
      Contact( "Siłownik_okien_otwieranie" )
      { S7_Templates := "SrcType := Real" } GE_Contact(in1 := "Wejscia_PLC".Temperatura_zewnetrzna, in2 := "Wejscia_PLC".Temperatura_wewnetrzna)
      Move(in := "Wejscia_PLC".Temperatura_zewnetrzna, out1 => "Wejscia_PLC".Temperatura_wewnetrzna)
   END_RUNG
   RUNG wire#powerrail
      { S7_Templates := "SrcType := Real" } LE_Contact(in1 := "Wejscia_PLC".Temperatura_wewnetrzna, in2 := 0.0)
      Move(in := 0.0, out1 => "Wejscia_PLC".Temperatura_wewnetrzna)
   END_RUNG
   // the same network as SCL:
   IF "Wejscia_PLC".Wewnetrzny_czujnik_CO2 <= "Wejscia_PLC".Zewnetrzny_czujnik_CO2 THEN
       "Wejscia_PLC".Wewnetrzny_czujnik_CO2 := "Wejscia_PLC".Zewnetrzny_czujnik_CO2;
   END_IF;
   IF "Wejscia_PLC".Czujnik_wilgotności_powietrza >= 100 THEN
       "Wejscia_PLC".Czujnik_wilgotności_powietrza := 100;
   END_IF;
   IF "Wejscia_PLC".Czujnik_wilgotności_gleby >= 100 THEN
       "Wejscia_PLC".Czujnik_wilgotności_gleby := 100;
   END_IF;
   IF "Wejscia_PLC".czujnik_wilgotnosci_zewnetrzny >= 100 THEN
       "Wejscia_PLC".czujnik_wilgotnosci_zewnetrzny := 100;
   END_IF;
   IF "Wejscia_PLC".Wewnetrzny_czujnik_CO2 >= 5000 THEN "Wejscia_PLC".Wewnetrzny_czujnik_CO2 := 5000; END_IF;
   IF "Wejscia_PLC".Zewnetrzny_czujnik_CO2 >= 5000 THEN "Wejscia_PLC".Wewnetrzny_czujnik_CO2 := 5000; END_IF;
   IF "Wejscia_PLC".Czujnik_natezenia_swiatła >= 1500 THEN
       "Wejscia_PLC".Czujnik_natezenia_swiatła := 1500;
   END_IF;
   IF "Wejscia_PLC".Czujnik_wilgotności_powietrza <= 0 THEN
       "Wejscia_PLC".Czujnik_wilgotności_powietrza := 0;
   END_IF;
   IF "Wejscia_PLC".Czujnik_wilgotności_gleby <= 0 THEN "Wejscia_PLC".Czujnik_wilgotności_gleby := 0; END_IF;
   IF "Wejscia_PLC".czujnik_wilgotnosci_zewnetrzny <= 0 THEN
       "Wejscia_PLC".czujnik_wilgotnosci_zewnetrzny := 0;
   END_IF;
   IF "Wejscia_PLC".Wewnetrzny_czujnik_CO2 <= 0 THEN "Wejscia_PLC".Wewnetrzny_czujnik_CO2 := 0; END_IF;
   IF "Wejscia_PLC".Zewnetrzny_czujnik_CO2 <= 0 THEN "Wejscia_PLC".Zewnetrzny_czujnik_CO2 := 0; END_IF;
   IF "Wejscia_PLC".Czujnik_natezenia_swiatła <= 0 THEN "Wejscia_PLC".Czujnik_natezenia_swiatła := 0; END_IF;
   IF "Wejscia_PLC".Stopien_zasloniecia_rolet >= 100 THEN
       "Wejscia_PLC".Stopien_zasloniecia_rolet := 100;
   END_IF;
   IF "Wejscia_PLC".Stopien_zasloniecia_rolet <= 0 THEN "Wejscia_PLC".Stopien_zasloniecia_rolet := 0; END_IF;
   IF "Wejscia_PLC".Temperatura_zewnetrzna >= 50.0 THEN "Wejscia_PLC".Temperatura_zewnetrzna := 50.0; END_IF;
   IF "Wejscia_PLC".Temperatura_wewnetrzna >= 50.0 THEN "Wejscia_PLC".Temperatura_wewnetrzna := 50.0; END_IF;
   IF "Siłownik_okien_otwieranie" AND ("Wejscia_PLC".Temperatura_zewnetrzna >= "Wejscia_PLC".Temperatura_wewnetrzna) THEN
       "Wejscia_PLC".Temperatura_wewnetrzna := "Wejscia_PLC".Temperatura_zewnetrzna;
   END_IF;
   IF "Wejscia_PLC".Temperatura_wewnetrzna <= 0.0 THEN "Wejscia_PLC".Temperatura_wewnetrzna := 0.0; END_IF;
END_REGION

REGION Network 20: symulacja predkosci wiatru
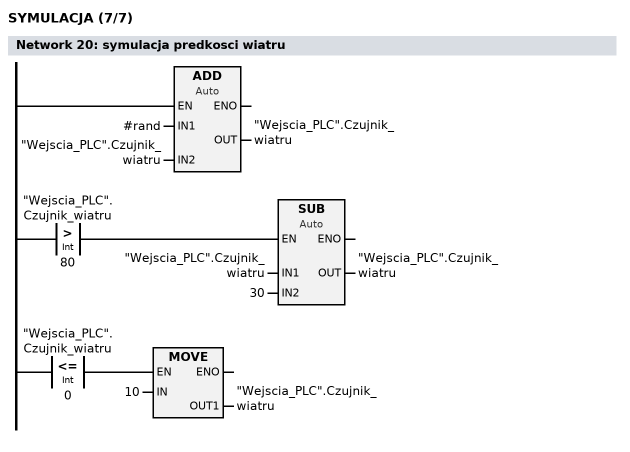
   RUNG wire#powerrail
      Add(in1 := #rand, in2 := "Wejscia_PLC".Czujnik_wiatru, out => "Wejscia_PLC".Czujnik_wiatru)
   END_RUNG
   RUNG wire#powerrail
      { S7_Templates := "SrcType := Int" } GT_Contact(in1 := "Wejscia_PLC".Czujnik_wiatru, in2 := 80)
      Sub(in1 := "Wejscia_PLC".Czujnik_wiatru, in2 := 30, out => "Wejscia_PLC".Czujnik_wiatru)
   END_RUNG
   RUNG wire#powerrail
      { S7_Templates := "SrcType := Int" } LE_Contact(in1 := "Wejscia_PLC".Czujnik_wiatru, in2 := 0)
      Move(in := 10, out1 => "Wejscia_PLC".Czujnik_wiatru)
   END_RUNG
   // the same network as SCL:
   "Wejscia_PLC".Czujnik_wiatru := #rand + "Wejscia_PLC".Czujnik_wiatru;
   IF "Wejscia_PLC".Czujnik_wiatru > 80 THEN
       "Wejscia_PLC".Czujnik_wiatru := "Wejscia_PLC".Czujnik_wiatru - 30;
   END_IF;
   IF "Wejscia_PLC".Czujnik_wiatru <= 0 THEN "Wejscia_PLC".Czujnik_wiatru := 10; END_IF;
END_REGION
END_FUNCTION

ORGANIZATION_BLOCK "Main"   // OB1, LAD, ProgramCycle
TITLE = "Main Program Sweep (Cycle)"
{ S7_Optimized_Access := 'TRUE' }
VERSION : 0.1
   VAR_INPUT
      Initial_Call : Bool;   // Initial call of this OB
      Remanence : Bool;   // =True, if remanent data are available
   END_VAR
   VAR_TEMP   // added for the SCL form of the ladder/FBD networks
      _w1 : Bool;
   END_VAR
BEGIN

REGION Network 1
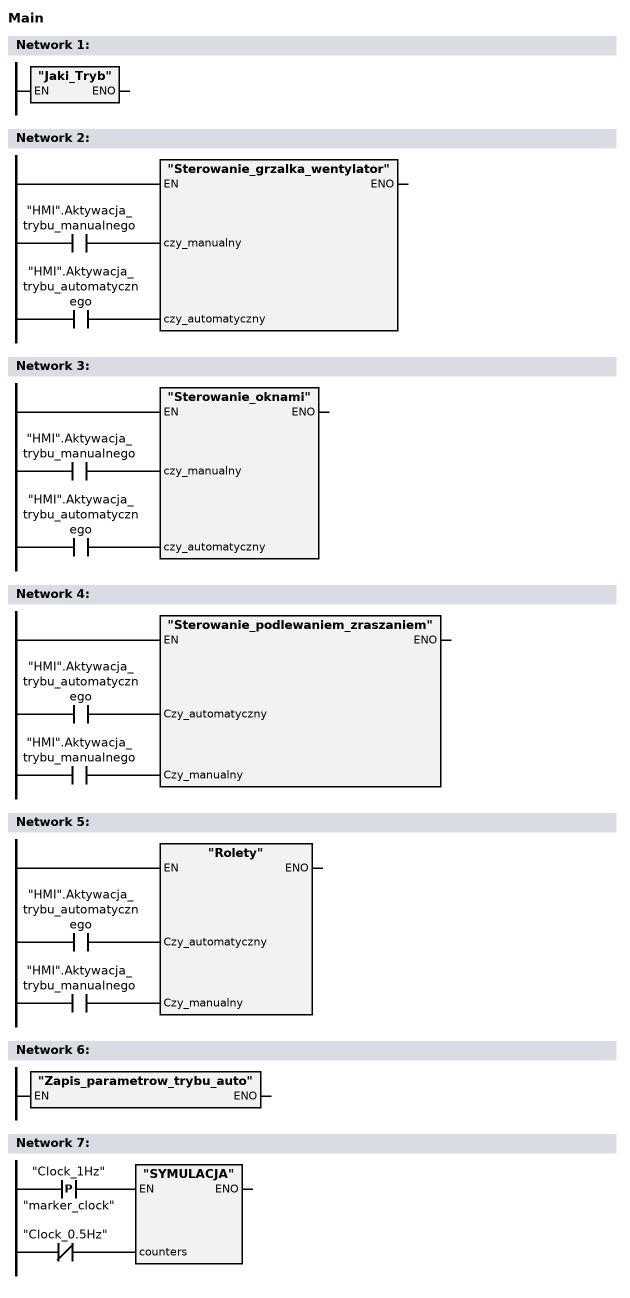
   RUNG wire#powerrail
      "Jaki_Tryb"()
   END_RUNG
   // the same network as SCL:
   "Jaki_Tryb"();
END_REGION

REGION Network 2
   RUNG wire#powerrail
      "Sterowanie_grzalka_wentylator"(czy_manualny := wire#w1, czy_automatyczny := wire#w2)
   END_RUNG
   RUNG wire#powerrail
      Contact( "HMI".Aktywacja_trybu_manualnego )
   END_RUNG wire#w1
   RUNG wire#powerrail
      Contact( "HMI".Aktywacja_trybu_automatycznego )
   END_RUNG wire#w2
   // the same network as SCL:
   "Sterowanie_grzalka_wentylator"(czy_manualny := "HMI".Aktywacja_trybu_manualnego,
                           czy_automatyczny := "HMI".Aktywacja_trybu_automatycznego);
END_REGION

REGION Network 3
   RUNG wire#powerrail
      "Sterowanie_oknami"(czy_manualny := wire#w1, czy_automatyczny := wire#w2)
   END_RUNG
   RUNG wire#powerrail
      Contact( "HMI".Aktywacja_trybu_manualnego )
   END_RUNG wire#w1
   RUNG wire#powerrail
      Contact( "HMI".Aktywacja_trybu_automatycznego )
   END_RUNG wire#w2
   // the same network as SCL:
   "Sterowanie_oknami"(czy_manualny := "HMI".Aktywacja_trybu_manualnego,
                       czy_automatyczny := "HMI".Aktywacja_trybu_automatycznego);
END_REGION

REGION Network 4
   RUNG wire#powerrail
      "Sterowanie_podlewaniem_zraszaniem"(Czy_automatyczny := wire#w1, Czy_manualny := wire#w2)
   END_RUNG
   RUNG wire#powerrail
      Contact( "HMI".Aktywacja_trybu_automatycznego )
   END_RUNG wire#w1
   RUNG wire#powerrail
      Contact( "HMI".Aktywacja_trybu_manualnego )
   END_RUNG wire#w2
   // the same network as SCL:
   "Sterowanie_podlewaniem_zraszaniem"(Czy_automatyczny := "HMI".Aktywacja_trybu_automatycznego,
                           Czy_manualny := "HMI".Aktywacja_trybu_manualnego);
END_REGION

REGION Network 5
   RUNG wire#powerrail
      "Rolety"(Czy_automatyczny := wire#w1, Czy_manualny := wire#w2)
   END_RUNG
   RUNG wire#powerrail
      Contact( "HMI".Aktywacja_trybu_automatycznego )
   END_RUNG wire#w1
   RUNG wire#powerrail
      Contact( "HMI".Aktywacja_trybu_manualnego )
   END_RUNG wire#w2
   // the same network as SCL:
   "Rolety"(Czy_automatyczny := "HMI".Aktywacja_trybu_automatycznego,
            Czy_manualny := "HMI".Aktywacja_trybu_manualnego);
END_REGION

REGION Network 6
   RUNG wire#powerrail
      "Zapis_parametrow_trybu_auto"()
   END_RUNG
   // the same network as SCL:
   "Zapis_parametrow_trybu_auto"();
END_REGION

REGION Network 7
   RUNG wire#powerrail
      P_Contact(operand := "Clock_1Hz", bit := "marker_clock")
      "SYMULACJA"(counters := wire#w1)
   END_RUNG
   RUNG wire#powerrail
      I_Contact( "Clock_0.5Hz" )
   END_RUNG wire#w1
   // the same network as SCL:
   #_w1 := "Clock_1Hz" AND NOT "marker_clock";   // rising edge of "Clock_1Hz"
   "marker_clock" := "Clock_1Hz";
   IF #_w1 THEN "SYMULACJA"(counters := NOT "Clock_0.5Hz"); END_IF;
END_REGION
END_ORGANIZATION_BLOCK

// folder: Archiwizacja_parametrow

FUNCTION "Archiwizacja_parametrow" : Void   // FC2, LAD
{ S7_Optimized_Access := 'TRUE' }
VERSION : 0.1
// Zapis parametrów do bloku DB odbywa się co pół godziny. Po uruchomieniu sterownika pierwszy zapis nie odbywa się od razu, aby wykres nie przedstawiał parametrów, które nie były jeszcze regulowane. Oczytane watosci zapisywane są w tablicach w bloku DB.
   VAR CONSTANT
      iterator : Int := 0;
   END_VAR
   VAR_TEMP   // added for the SCL form of the ladder/FBD networks
      _w1 : Bool;
   END_VAR
BEGIN

REGION Network 1
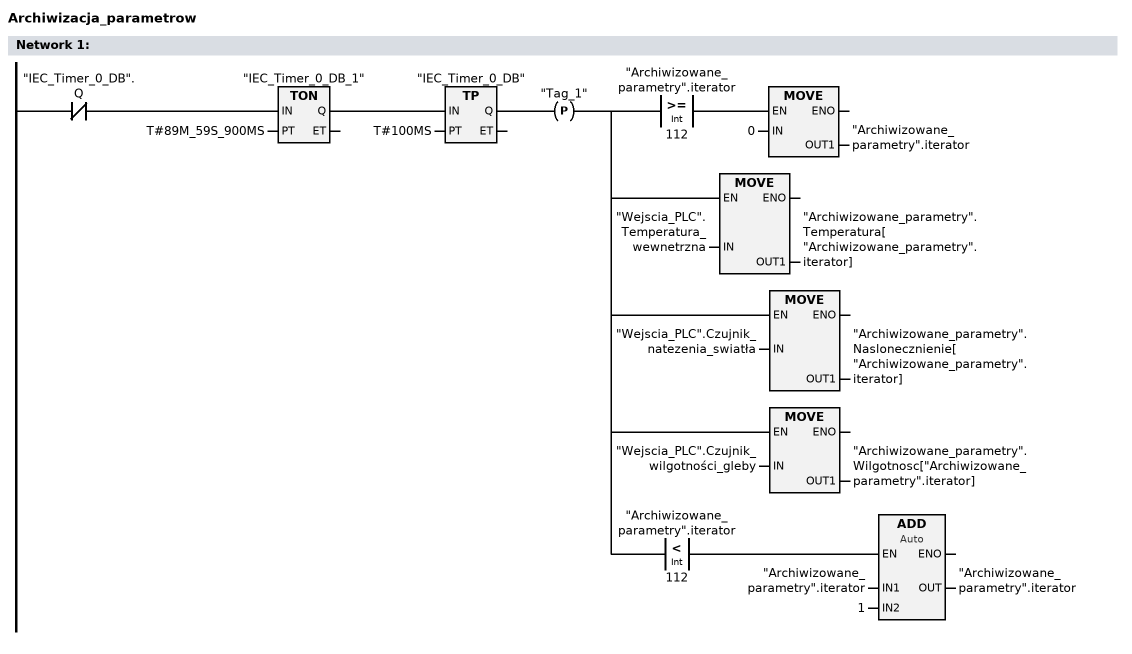
   "IEC_Timer_0_DB_1".TON(IN := NOT "IEC_Timer_0_DB".Q, PT := T#89M_59S_900MS);
   "IEC_Timer_0_DB".TP(IN := "IEC_Timer_0_DB_1".Q, PT := T#100MS);
   #_w1 := "IEC_Timer_0_DB".Q AND NOT "Tag_1";   // rising edge
   "Tag_1" := "IEC_Timer_0_DB".Q;
   IF #_w1 AND ("Archiwizowane_parametry".iterator >= 112) THEN
       "Archiwizowane_parametry".iterator := 0;
   END_IF;
   IF #_w1 THEN
       "Archiwizowane_parametry".Temperatura["Archiwizowane_parametry".iterator] := "Wejscia_PLC".Temperatura_wewnetrzna;
       "Archiwizowane_parametry".Naslonecznienie["Archiwizowane_parametry".iterator] := "Wejscia_PLC".Czujnik_natezenia_swiatła;
       "Archiwizowane_parametry".Wilgotnosc["Archiwizowane_parametry".iterator] := "Wejscia_PLC".Czujnik_wilgotności_gleby;
   END_IF;
   IF #_w1 AND ("Archiwizowane_parametry".iterator < 112) THEN
       "Archiwizowane_parametry".iterator := "Archiwizowane_parametry".iterator + 1;
   END_IF;
END_REGION
END_FUNCTION

// folder: LGF/4 Math operations

FUNCTION "LGF_RandomRange_Real" : Real   // FC10014, SCL
TITLE = LGF_RandomRange_Real
{ S7_Optimized_Access := 'TRUE' }
AUTHOR : Siemens_Digital_Industries
FAMILY : LGF
NAME : LGF_RandomRange_Real
// This function generates random numbers in defined limits (Datatype Real)
   VAR_INPUT
      minValue : Real;   // minimal Value random can reach / Minimum value of the range of the random number
      maxValue : Real;   // maximal Value random can reach / Maximum value of the range of the random number
   END_VAR
   VAR_OUTPUT
      error : Bool;   // Error if true
      status : Word;   // Status of the function
      subfunctionStatus : Word;   // Status or return value of called FB's, FCs and system blocks
   END_VAR
   VAR_TEMP
      tempTime : DTL;   // System time
      tempNanoSecondInDWord : DWord;   // UDINT converted to DWORD for access to individual bytes
      tempTimeStatus : Word;   // Status of the instruction RD_SYS_T
      tempRandomValue : DWord;   // Random-start-value
      tempNormReal : Real;   // normalized value
   END_VAR
   // Ret_Val : Returns random Real number in predefined range
   VAR CONSTANT
      ZERO : Real := 0.0;   // Zero value in case of error
      MAX_UDINT : UDInt := 4294967295;   // Maximum UDINT value
      SUB_STATUS_NO_ERROR : Word := 16#0000;   // Status: sub function call ends without error
      STATUS_FINISHED_NO_ERROR : Word := 16#0000;   // Status: Execution finished without errors
      ERR_MAX_LESS_MIN : Word := 16#8200;   // Error: The maximum limit number is smaller than the minimum limit number
      ERR_RD_SYS_T : Word := 16#8600;   // Error: System function Read system time returned an error
   END_VAR
BEGIN
   REGION Block info header
     //=============================================================================
     // SIEMENS AG / (c)Copyright 2017
     //-----------------------------------------------------------------------------
     // Title:            LGF_RandomRange_Real
     // Comment/Function: This function generates random numbers in defined limits (Datatype Real)
     // Library/Family:   LGF(Library General Functions)
     // Author:           Siemens Digital Industry Support
     // Tested with:      S7-PLCSIM Advanced V2.0 SP1
     // Engineering:      TIA Portal V15 Update 2
     // Restrictions:     ENO disabled - error handling done by error and status
     // Requirements:     PLC (S7-1200 / S7-1500)
     //-------------------------------------------------------------------------------
     // Change log table:
     // Version  | Date       | Expert in charge       | Changes applied
     //----------|------------|------------------------|------------------------------
     // 01.00.00 19.08.2015  Siemens Industry Online Support
     //                      First released version
     // 01.00.01 02.01.2017  Siemens Industry Online Support
     //                      Upgrade: TIA Portal V14 Update 1
     // 01.00.02 02.03.2017  Siemens Industry Online Support
     //                      Bugfix: FC number
     // 01.00.03 17.08.2018  Siemens Industry Online Support
     //                      Upgrade: TIA V15 Update 2
     // 01.00.04 23.11.2018  Siemens Industry Online Support
     //                      Upgrade: TIA V15.1
     // 01.01.00 13.11.2019  Siemens Industry Presales Support
     //                      Renamed from "LGF_RandomReal" to "LGF_RandomRange_Real"
     //                      Regions, commens and costants are added
     // 03.00.00 23.04.2020  Siemens Industry Support
     //                      Set version to V3.0.0, harmonize the version of the whole library
     //=============================================================================
   END_REGION

   REGION Validation
     // Check if the maximal Value is less than the minimal value
     IF (#minValue > #maxValue) THEN
       #error := true;
       #status := #ERR_MAX_LESS_MIN;
       #subfunctionStatus := #SUB_STATUS_NO_ERROR;
       #LGF_RandomRange_Real := #ZERO;
       RETURN;
     END_IF;

     // Read system time
     #tempTimeStatus := INT_TO_WORD(RD_SYS_T(#tempTime));

     // Check return variable for error
     IF (#tempTimeStatus <> #SUB_STATUS_NO_ERROR) THEN
       #error := true;
       #status := #ERR_RD_SYS_T;
       #subfunctionStatus := #tempTimeStatus;
       #LGF_RandomRange_Real := #ZERO;
       RETURN;
     END_IF;
   END_REGION

   REGION Calculating random number
     // Converting to double word so individual bytes can be addressed
     #tempNanoSecondInDWord := UDINT_TO_DWORD(#tempTime.NANOSECOND);

     // Calculate a random-start-value depending on the time
     #tempRandomValue.%B3 := #tempNanoSecondInDWord.%B0;
     #tempRandomValue.%B2 := #tempNanoSecondInDWord.%B1;
     #tempRandomValue.%B1 := #tempNanoSecondInDWord.%B2;
     #tempRandomValue.%B0 := #tempNanoSecondInDWord.%B3;

     // Norm the calculated random number: 0.0 <= #tempNormReal <= 1.0
     #tempNormReal := UDINT_TO_REAL(DWORD_TO_UDINT(#tempRandomValue)) / UDINT_TO_REAL(#MAX_UDINT);

     // Scale the tempNormReal to be in the range of maxValue and minValue
     #LGF_RandomRange_Real := ((#tempNormReal * (#maxValue - #minValue) + (#minValue)));

     #error := false;
     #status := #STATUS_FINISHED_NO_ERROR;
     #subfunctionStatus := #SUB_STATUS_NO_ERROR;
     // ENO mechanism is not used
     ENO := TRUE;
   END_REGION
END_FUNCTION

// ===== PLC "PLC_Web_server"  CPU 1518-4 PN/DP =====

VAR_GLOBAL   // PLC tag table "Default tag table"
   "err" AT %MW1 : Int;
   "tag1" AT %M6.0 : Bool;
END_VAR

DATA_BLOCK "Wejscia_PLC"   // DB2
{ S7_Optimized_Access := 'TRUE' }
VERSION : 0.1
   VAR
      Czujnik_wilgotności_powietrza : Int;   // Czujnik wilgotności powietrza w szklarni
      Czujnik_wilgotności_gleby : Int;   // Czujnik wilgotności gleby w szklarni
      Temperatura_wewnetrzna : Real;   // Temperatura wewnątrz szklarni
      Czujnik_natezenia_swiatła : Int;   // Czujnik natężenia światła wewnątrz szklarni
      Wewnetrzny_czujnik_CO2 : Int;   // Czujnik stężenia dwutlenku węgla w szklarni
      Stopien_zasloniecia_rolet : Int;   // Stopień zasłonięcia rolet w szklarni (przyjęty przedział 0-100%)
   END_VAR
BEGIN
END_DATA_BLOCK

// folder: Archiwizacja_parametrow

DATA_BLOCK "Archiwizowane_parametry"   // DB4
{ S7_Optimized_Access := 'TRUE' }
VERSION : 0.1
   VAR
      Temperatura : Array[0..111] of Real;
      Wilgotnosc : Array[0..111] of Int;
      Naslonecznienie : Array[0..111] of Int;
      iterator : Int := 0;   // Iterator służący do zapisu danych w odpowiednich komórkach tablicy.
   END_VAR
BEGIN
   Naslonecznienie[0] := 0;
   Naslonecznienie[1] := 0;
END_DATA_BLOCK

// folder: (top level)

ORGANIZATION_BLOCK "Main"   // OB1, LAD, ProgramCycle
TITLE = "Main Program Sweep (Cycle)"
{ S7_Optimized_Access := 'TRUE' }
VERSION : 0.1
   VAR_INPUT
      Initial_Call : Bool;   // Initial call of this OB
      Remanence : Bool;   // =True, if remanent data are available
   END_VAR
BEGIN

REGION Network 1
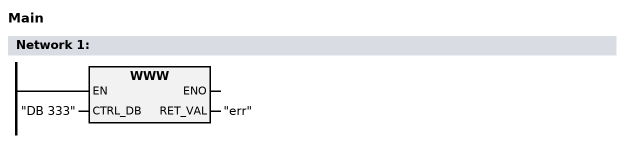
   "err" := WWW(CTRL_DB := "DB 333");
END_REGION
END_ORGANIZATION_BLOCK

(* ===== HMI "HMI_RT_3" =====
system functions are stored by id; their names below are inferred from use
connection "HMI_Connection_4": ETHERNET, SMART_S7_1200_OMS

HMI tags "Default tag table"
   "AlwaysTRUE" : Bool = PLC AlwaysTRUE AT %M1.2, 1 s
   "Grzałka" : Bool = PLC Grzałka AT %Q0.0, 1 s
   "HMI_Aktywacja_trybu_automatycznego" : Bool = PLC HMI.Aktywacja_trybu_automatycznego, 1 s
   "HMI_Aktywacja_trybu_Receptur" : Bool = PLC HMI.Aktywacja_trybu_Receptur, 1 s
   "HMI_Aktywacja_trybu_zapis_Receptur" : Bool = PLC HMI.Aktywacja_trybu_zapis_Receptur, 1 s
   "HMI_Reset_Trybow" : Bool = PLC HMI.Reset_Trybow, 1 s
   "Pompa_podlewanie" : Bool = PLC Pompa_podlewanie AT %Q1.0, 1 s
   "Pompa_zraszacze" : Bool = PLC Pompa_zraszacze AT %Q0.2, 1 s
   "Tag_ScreenNumber" : Int = PLC HMI.Numer_ekranu_HMI AT %MD0, 100 ms
   "Tryb_auto_parametry_Naslonecznienie" : Int = PLC Tryb_auto_parametry.Naslonecznienie, 1 s
   "Tryb_auto_parametry_Stezenie_co2" : Int = PLC Tryb_auto_parametry.Stezenie_co2, 1 s
   "Tryb_auto_parametry_System_okien" : Bool = PLC Tryb_auto_parametry.System_okien, 1 s
   "Tryb_auto_parametry_Temperatura" : Real = PLC Tryb_auto_parametry.Temperatura, 1 s
   "Tryb_auto_parametry_Wilgotnosc_gleby" : Int = PLC Tryb_auto_parametry.Wilgotnosc_gleby, 1 s
   "Tryb_auto_parametry_Wilgotnosc_powietrza" : Int = PLC Tryb_auto_parametry.Wilgotnosc_powietrza, 1 s
   "Wentylator" : Bool = PLC Wentylator AT %Q0.1, 1 s

HMI tags "Z_PLC"
   "Czujnik_wilgotności_powietrza" : Int = PLC Wejscia_PLC.Czujnik_wilgotności_powietrza, 500 ms
   "Temperatura_wewnetrzna" : Real = PLC Wejscia_PLC.Temperatura_wewnetrzna, 500 ms
   "Czujnik_natezenia_światła" : Int = PLC Wejscia_PLC.Czujnik_natezenia_swiatła, 500 ms
   "Czujnik_wilgotności_gleby" : Int = PLC Wejscia_PLC.Czujnik_wilgotności_gleby, 500 ms
   "Wewnetrzny_czujnik_CO2" : Int = PLC Wejscia_PLC.Wewnetrzny_czujnik_CO2, 500 ms
   "Czujnik_wiatru" : Int = PLC Wejscia_PLC.Czujnik_wiatru, 500 ms
   "Stopien_zasloniecia_rolet" : Int = PLC Wejscia_PLC.Stopien_zasloniecia_rolet, 1 s
   "Zewnetrzny_czujnik_CO2" : Int = PLC Wejscia_PLC.Zewnetrzny_czujnik_CO2 AT %DB1.DBW0, 1 s
   "Temperatura_zewnetrzna" : Real = PLC Wejscia_PLC.Temperatura_zewnetrzna AT %DB1.DBW0, 1 s

HMI tags "Do_PLC"
   "System_okien_auto" : Bool = PLC HMI.System_okien_auto, 500 ms
   "Stopien_zasloniecia_rolet_manual" : Int = PLC HMI.Stopien_zasloniecia_rolet_manual, 100 ms
   "Przycisk_zraszania_manual" : Bool = PLC HMI.Przycisk_zraszacze_manual AT %Q0.2, 100 ms
   "Przycisk_wentylacja_manual" : Bool = PLC HMI.Przycisk_wentylacja_manual AT %Q0.1, 100 ms
   "Przycisk_grzanie_manual" : Bool = PLC HMI.Przycisk_grzanie_manual AT %Q0.0, 100 ms
   "Otwarcie_okien_man" : Bool = PLC HMI.Otwarcie_okien_manual AT %DB1.DBW0, 100 ms
   "Temperatura_auto" : Real = PLC HMI.Temperatura_auto, 500 ms
   "Naslonecznienie_auto" : Int = PLC HMI.Naslonecznienie_auto AT %DB1.DBW0, 500 ms
   "Wilgotnosc_powietrza_auto" : Int = PLC HMI.Wilgotnosc_powietrza_auto AT %DB1.DBW0, 500 ms
   "Wilgotnosc_gleby_auto" : Int = PLC HMI.Wilgotnosc_gleby_auto AT %DB1.DBW0, 500 ms
   "Przycisk_zatwierdz_auto" : Bool = PLC HMI.Przycisk_zatwierdz_auto AT %DB1.DBW0, 100 ms
   "nazwa_receptury" : String[254] = PLC HMI.nazwa_receptury AT %DB1.DBX0.0, 500 ms
   "przycisk_zatwierdz_zapis_receptury" : Bool = PLC HMI.Przycisk_zatwierdz_zapis_receptury AT %DB1.DBX0.0, 500 ms
   "HMI_Przycisk_zatwierdz_wybor_receptury" : Bool = PLC HMI.Przycisk_zatwierdz_wybor_receptury AT %DB1.DBX0.0, 500 ms
   "Przycisk_podlewania_manual" : Bool = PLC HMI.Przycisk_podlewanie_manual AT %Q0.2, 100 ms
   "Poziom_CO2_auto" : Int = PLC HMI.Poziom_CO2_auto AT %DB1.DBX0.0, 1 s

analog alarms
   3: 'Podmuchy wiatru osiągają wartości powyżej 35 km/h, system automatyczny zamyka okna.', class Warnings, trigger "Czujnik_wiatru"
   2: 'Temperatura powyżej 35 stopni / Temperatura powyżej 35 stopni, zaleca się wyłączenie grzania.', class Warnings, trigger "Temperatura_wewnetrzna"
   5: 'Temperatura powyżej 45 stopni, NIEZWŁOCZNIE SPRAWDŹ DZIAŁANIE GRZAŁKI, TERMOMETRU LUB WENTYLATORA. / Temperatura powyżej 45 stopni, NIEZWŁOCZNIE SPRAWDŹ DZIAŁANIE GRZAŁKI, TERMOMETRU LUB WENTYLATORA. JEŚLI TEMPERATURA NIE SPADA ZALECA SIĘ EWAKUOWAĆ WSZYSTKICH PRZEBYWAJĄCYCH W POMIESZCZENIU', class Errors, trigger "Temperatura_wewnetrzna"
   4: 'Stężenie CO2 ma powyżej 5000 jednostek. NIEZWŁOCZNIE OTWORZ OKNA ORAZ ZAŁĄCZ WENTYLATOR, NASTĘPNIE NALEŻY EWAKUOWAĆ WSZYSTKUCH ZNAJDUJĄCYCH SIĘ W POMIESZCZENIU / Stężenie CO2 ma powyżej 5000 jednostek. NIEZWŁOCZNIE OTWORZ OKNA ORAZ ZAŁĄCZ WENTYLATOR, NASTĘPNIE NALEŻY EWAKUOWAĆ WSZYSTKUCH ZNAJDUJĄCYCH SIĘ W POMIESZCZENIU', class Errors, trigger "Wewnetrzny_czujnik_CO2"
   1: 'Stężenie CO2 ma powyżej 3000 jednostek / Stężenie CO2 ma powyżej 3000 jednostek, dłużesze przebywanie w takim środowisku może być szkodliwe dla człowieka. Zalecane jest włączenie wentylacji lub otworzenie okien.', class Warnings, trigger "Wewnetrzny_czujnik_CO2"

text list "receptury": 0..1 ''

recipe "Receptura_nr1": Temperatura <- "Tryb_auto_parametry_Temperatura", Wilgotność Powietrza <- "Tryb_auto_parametry_Wilgotnosc_powietrza", Wilgotność gleby <- "Tryb_auto_parametry_Wilgotnosc_gleby", System okien <- "Tryb_auto_parametry_System_okien", Stężenie CO2 <- "Tryb_auto_parametry_Stezenie_co2", Nasłonecznienie <- "Tryb_auto_parametry_Naslonecznienie"

screen "tryb_manualny" 800x480
   on GenerateScreen: SetTag("Tag_ScreenNumber", 2)
   TextField "Text field_1" at 295,7 size 223x34; Text 'TRYB MANUALNY'
   TextField "Text field_4" at 512,155 size 171x61; Text 'STOPIEŃ OTWARCIA OKIEN OTWIERANIE OKIEN'
   Button "Button_4" at 518,261 size 80x70; TextOff 'PODLEWANIE'
      on Click: InvertBit("Przycisk_podlewania_manual")
   Button "Button_5" at 611,261 size 80x70; TextOff 'GRZANIE'
      on Click: InvertBit("Przycisk_grzanie_manual")
   Button "Button_6" at 701,261 size 80x70; TextOff 'WENTYLACJA'
      on Click: InvertBit("Przycisk_wentylacja_manual")
   GraphicView "Graphic view_1" at 710,356 size 60x60; Picture "fan_4829316"
      Visibility <- "Wentylator"
   GraphicView "Graphic view_6" at 622,356 size 60x60; Picture "heater_4463010"
      Visibility <- "Grzałka"
   GraphicView "Graphic view_7" at 527,356 size 64x60; Picture "irrigation_18631825"
      Visibility <- "Pompa_podlewanie"
   GraphicView "Graphic view_9" at 710,356 size 60x60; Picture "fan_off"
      Visibility <- "Wentylator"
   GraphicView "Graphic view_10" at 622,356 size 60x60; Picture "heater_off"
      Visibility <- "Grzałka"
   GraphicView "Graphic view_11" at 527,356 size 64x60; Picture "irrigation_off"
      Visibility <- "Pompa_podlewanie"
   Button "Button_14" at 6,7 size 43x43; TextOff 'DOM'; PictureOff "home_1"
      on Click: ActivateScreen("Root screen", 0)
   Button "Button_1" at 740,0 size 60x60; TextOff 'Text'; PictureOff "Back_arrow"
      on Click: function_efd93a16()
   Circle "Circle_1" at 541,428 size 42x42
      Visibility <- "Pompa_podlewanie"
   Circle "Circle_4" at 541,428 size 42x42
      Visibility <- "Pompa_podlewanie"
   Circle "Circle_2" at 631,428 size 42x42
      Visibility <- "Grzałka"
   Circle "Circle_5" at 631,428 size 42x42
      Visibility <- "Grzałka"
   Circle "Circle_3" at 720,428 size 41x41
      Visibility <- "Wentylator"
   Circle "Circle_6" at 720,428 size 41x41
      Visibility <- "Wentylator"
   TextField "Text field_8" at 405,71 size 117x61; Text 'STOPIEŃ OTWARCIA OKIEN STOPIEŃ ZASŁONIECIA ROLET'
   Bar "Bar_6" at 624,82 size 165x66; MinimumValue 0; MaximumValue 100
      ProcessValue <- "Stopien_zasloniecia_rolet_manual"
   Button "Button_3" at 530,114 size 80x50; TextOff '+ / ODSŁOŃ'
      on Click: function_b9b71300("Stopien_zasloniecia_rolet_manual", 5)
   Button "Button_7" at 530,60 size 80x50; TextOff '- / ZASŁOŃ'
      on Press: function_dd21b452("Stopien_zasloniecia_rolet_manual", 5)
   Button "Button_2" at 425,261 size 80x70; TextOff 'PODLEWANIE / MIKROZRASZANIE'
      on Click: InvertBit("Przycisk_zraszania_manual")
   GraphicView "Graphic view_2" at 434,356 size 60x60; Picture "sprinkler_4552152"
      Visibility <- "Pompa_zraszacze"
   GraphicView "Graphic view_3" at 434,356 size 60x60; Picture "sprinkler"
      Visibility <- "Pompa_zraszacze"
   Circle "Circle_7" at 443,428 size 42x42
      Visibility <- "Pompa_zraszacze"
   Circle "Circle_8" at 443,428 size 42x42
      Visibility <- "Pompa_zraszacze"
   Switch "Switch_1" at 499,199 size 209x37; TextOn 'OTWARTE'; CaptionText 'Switch'; TextOff 'ZAMKNIĘTE'
      ProcessValue <- "Otwarcie_okien_man"
   TextField "Text field_3" at 11,375 size 166x23; Text 'SZYBKOŚĆ WIATRU'
   IOField "I/O field_3" at 62,407 size 70x65; FormatPattern 999
      ProcessValue <- "Czujnik_wiatru"
   IOField "I/O field_1" at 48,189 size 101x32; FormatPattern 99999
      ProcessValue <- "Czujnik_natezenia_światła"
   TextField "Text field_15" at 129,408 size 52x72; Text 'Km h'
   IOField "I/O field_2" at 44,292 size 83x65; FormatPattern 9999
      ProcessValue <- "Wewnetrzny_czujnik_CO2"
   TextField "Text field_11" at 118,301 size 69x39; Text 'ppm'
   TextField "Text field_5" at 14,148 size 204x23; Text 'INSOLATION / NASŁONECZNIENIE / SONNENEINSTRAHLUNG'
   IOField "I/O field_8" at 58,95 size 93x40; FormatPattern 99.99
      ProcessValue <- "Temperatura_wewnetrzna"
   TextField "Text field_20" at 30,56 size 137x42; Text 'TEMPERATURA TEMPERATURA WEWNTĘTRZNA'
   TextField "Text field_7" at 200,375 size 175x23; Text 'WILGOTNOŚĆ GLEBY'
   IOField "I/O field_5" at 248,293 size 83x65; FormatPattern 9999
      ProcessValue <- "Zewnetrzny_czujnik_CO2"
   IOField "I/O field_4" at 266,174 size 69x65; FormatPattern 999
      ProcessValue <- "Czujnik_wilgotności_powietrza"
   IOField "I/O field_6" at 261,405 size 68x65; FormatPattern 999
      ProcessValue <- "Czujnik_wilgotności_gleby"
   TextField "Text field_12" at 324,182 size 47x46; Text '%'
   TextField "Text field_13" at 321,416 size 47x46; Text '%'
   TextField "Text field_16" at 326,292 size 69x39; Text 'ppm'
   IOField "I/O field_9" at 248,85 size 97x65; FormatPattern 99.99
      ProcessValue <- "Temperatura_zewnetrzna"
   TextField "Text field_23" at 333,90 size 46x46; Text '°C'
   TextField "Text field_22" at 229,57 size 132x42; Text 'TEMPERATURA TEMPERATURA ZEWNĘTRZNA'
   TextField "Text field_9" at 229,256 size 123x42; Text 'STĘŻENIE CO2 ZEWNĘTRZNE STĘŻENIE CO2'
   TextField "Text field_6" at 180,143 size 223x42; Text 'WILGOTNOŚĆ POWIETRZA WILGOTNOŚĆ POWIETRZA'
   TextField "Text field_14" at 140,170 size 47x72; Text 'W m²'
   TextField "Text field_21" at 141,90 size 46x46; Text '°C'
   GraphicView "Graphic view_4" at 419,176 size 60x60; Picture "window_11250237"
   GraphicView "Graphic view_5" at 197,182 size 50x50; Picture "sensor_4212519"
   GraphicView "Graphic view_8" at 4,182 size 50x50; Picture "sensor_4212513"
   GraphicView "Graphic view_12" at 3,87 size 50x50; Picture "Thermometer_icon"
   GraphicView "Graphic view_13" at 199,87 size 50x50; Picture "Thermometer_icon"
   GraphicView "Graphic view_14" at 3,302 size 40x40; Picture "sensor_2828470"
   GraphicView "Graphic view_15" at 197,300 size 40x40; Picture "sensor_2828470"
   GraphicView "Graphic view_16" at 198,412 size 50x50; Picture "soil-sensor_11298794"
   GraphicView "Graphic view_17" at 3,416 size 50x50; Picture "anemometer_1113716"
   TextField "Text field_2" at 27,256 size 124x42; Text 'STĘŻENIE CO2 WEWNĘTRZNE STĘŻENIE CO2'

screen "tryb_automatyczny" 800x480
   on GenerateScreen: SetTag("Tag_ScreenNumber", 1)
   IOField "I/O field_1" at 67,322 size 57x40; FormatPattern 99.9
      ProcessValue <- "Temperatura_wewnetrzna"
   Button "Button_1" at 745,0 size 55x55; TextOff 'WRÓĆ'; PictureOff "Back_arrow"
      on Click: function_efd93a16()
   Button "Button_2" at 373,382 size 416x89; TextOff 'ZATWIERDŹ'
      on Click: ResetBit("HMI_Reset_Trybow"); SetBit("HMI_Aktywacja_trybu_automatycznego"); ActivateScreen("praca", 0)
   Bar "Bar_1" at 7,110 size 50x250; MinimumValue 0; MaximumValue 45
      ProcessValue <- "Temperatura_auto"
   TextField "Text field_2" at 1,71 size 132x23; Text 'TEMPERATURA'
   Bar "Bar_2" at 170,111 size 50x250; MinimumValue 0; MaximumValue 100
      ProcessValue <- "Wilgotnosc_powietrza_auto"
   TextField "Text field_3" at 165,68 size 122x42; Text 'WOLGOTNOŚĆ POWIETRZA WILGOTNOŚĆ POWIETRZA'
   Button "Button_3" at 71,115 size 75x45; TextOff '+ / +0.5 °C'
      on Press: function_dd21b452("Temperatura_auto", 0.5)
   Button "Button_7" at 71,183 size 75x45; TextOff '- / -0.5 °C'
      on Press: function_b9b71300("Temperatura_auto", 0.5)
   IOField "I/O field_2" at 67,251 size 62x40; FormatPattern 99.9
      ProcessValue <- "Temperatura_auto"
   TextField "Text field_11" at 122,260 size 23x22; Text '°C'
   TextField "Text field_9" at 122,333 size 23x22; Text '°C'
   Bar "Bar_4" at 335,111 size 50x250; MinimumValue 0; MaximumValue 100
      ProcessValue <- "Wilgotnosc_gleby_auto"
   TextField "Text field_10" at 332,65 size 122x42; Text 'WOLGOTNOŚĆ GLEBY WILGOTNOŚĆ GLEBY'
   Button "Button_8" at 398,132 size 65x40; TextOff '+ / +2%'
      on Click: function_dd21b452("Wilgotnosc_gleby_auto", 2)
   Button "Button_9" at 398,181 size 65x40; TextOff '- / -2%'
      on Click: function_b9b71300("Wilgotnosc_gleby_auto", 2)
   IOField "I/O field_5" at 402,255 size 60x40; FormatPattern 999
      ProcessValue <- "Wilgotnosc_gleby_auto"
   IOField "I/O field_6" at 404,325 size 58x40; FormatPattern 999
      ProcessValue <- "Czujnik_wilgotności_gleby"
   TextField "Text field_12" at 385,243 size 101x22; Text 'USTAWIONA'
   TextField "Text field_13" at 389,314 size 86x22; Text 'AKTUALNA'
   TextField "Text field_14" at 439,264 size 23x22; Text '%'
   TextField "Text field_15" at 439,335 size 23x22; Text '%'
   Button "Button_10" at 229,126 size 65x40; TextOff '+ / +5%'
      on Click: function_dd21b452("Wilgotnosc_powietrza_auto", 5)
   Button "Button_11" at 229,186 size 65x40; TextOff '- / -5%'
      on Click: function_b9b71300("Wilgotnosc_powietrza_auto", 5)
   IOField "I/O field_4" at 234,248 size 66x40; FormatPattern 999
      ProcessValue <- "Wilgotnosc_powietrza_auto"
   IOField "I/O field_7" at 236,320 size 62x40; FormatPattern 999
      ProcessValue <- "Czujnik_wilgotności_powietrza"
   TextField "Text field_16" at 223,235 size 101x22; Text 'USTAWIONA'
   TextField "Text field_17" at 223,306 size 86x22; Text 'AKTUALNA'
   TextField "Text field_18" at 275,257 size 23x22; Text '%'
   TextField "Text field_19" at 275,328 size 23x22; Text '%'
   Button "Button_14" at 4,7 size 45x45; TextOff 'DOM'; PictureOff "home_1"
      on Click: ActivateScreen("Root screen", 0)
   TextField "Text field_4" at 143,381 size 128x23; Text 'SYSTEM OKIEN'
   Switch "Switch_1" at 106,410 size 216x46; TextOn 'ON'; CaptionText 'Switch'; TextOff 'OFF'
      ProcessValue <- "System_okien_auto"
   GraphicView "Graphic view_1" at 129,70 size 40x40; Picture "Thermometer_icon"
   GraphicView "Graphic view_2" at 281,68 size 40x40; Picture "sensor_4212519"
   TextField "Text field_5" at 60,309 size 86x22; Text 'AKTUALNA'
   TextField "Text field_6" at 57,237 size 101x22; Text 'USTAWIONA'
   GraphicView "Graphic view_3" at 443,71 size 40x40; Picture "soil-sensor_11298794"
   TextField "Text field_1" at 255,4 size 291x47; Text 'TRYB AUTOMATYCZNY'
   Bar "Bar_3" at 496,111 size 50x250; MinimumValue 0; MaximumValue 1500
      ProcessValue <- "Naslonecznienie_auto"
   TextField "Text field_7" at 492,55 size 154x40; Text 'WOLGOTNOŚĆ GLEBY NASŁONECZNIENIE'
   GraphicView "Graphic view_4" at 585,86 size 40x40; Picture "sensor_4212513"
   Button "Button_4" at 553,131 size 82x43; TextOff '+ +50 W m'
      on Click: function_dd21b452("Naslonecznienie_auto", 50)
   Button "Button_5" at 554,186 size 82x43; TextOff '- -50 W m'
      on Click: function_b9b71300("Naslonecznienie_auto", 50)
   IOField "I/O field_3" at 561,254 size 61x40; FormatPattern 9999
      ProcessValue <- "Naslonecznienie_auto"
   TextField "Text field_8" at 545,242 size 101x22; Text 'USTAWIONA / USTAWIONE'
   IOField "I/O field_8" at 563,325 size 62x40; FormatPattern 9999
      ProcessValue <- "Czujnik_natezenia_światła"
   TextField "Text field_20" at 549,313 size 86x22; Text 'AKTUALNA / AKTUALNE'
   TextField "Text field_23" at 616,150 size 32x18; Text '2'
   TextField "Text field_24" at 614,205 size 32x18; Text '2'
   Bar "Bar_5" at 656,111 size 45x250; MinimumValue 400; MaximumValue 950
      ProcessValue <- "Poziom_CO2_auto"
   TextField "Text field_21" at 656,65 size 128x23; Text 'SYSTEM OKIEN / POZIOM CO2'
   IOField "I/O field_9" at 723,254 size 66x40; FormatPattern 999
      ProcessValue <- "Poziom_CO2_auto"
   TextField "Text field_22" at 699,216 size 101x22; Text 'USTAWIONA / USTAWIONE'
   IOField "I/O field_10" at 723,333 size 62x40; FormatPattern 999
      ProcessValue <- "Wewnetrzny_czujnik_CO2"
   TextField "Text field_25" at 708,314 size 86x22; Text 'AKTUALNA'
   Button "Button_6" at 714,134 size 73x40; TextOff '+ / +25ppm'
      on Click: function_dd21b452("Poziom_CO2_auto", 25)
   Button "Button_12" at 714,186 size 73x40; TextOff '+ / -25ppm'
      on Click: function_b9b71300("Poziom_CO2_auto", 25)
   GraphicView "Graphic view_5" at 754,83 size 40x40; Picture "sensor_2828470"
   GraphicView "Graphic view_6" at 17,400 size 55x55; Picture "window_11250237"

screen "Symulacja_czujnikow" 800x480
   TextField "Text field_1" at 12,58 size 252x23; Text 'Czujnik Wilgotności powietrza'
   TextField "Text field_2" at 306,58 size 214x23; Text 'Czujnik Wilgotności gleby'
   TextField "Text field_3" at 32,202 size 202x23; Text 'Termometr wewnętrzny'
   TextField "Text field_4" at 323,202 size 197x23; Text 'Termometr zewnętrzny'
   TextField "Text field_5" at 566,58 size 216x23; Text 'Czujnik natężenia światła'
   TextField "Text field_6" at 607,202 size 124x23; Text 'Czujnik wiatru'
   TextField "Text field_7" at 27,346 size 208x23; Text 'Wewnętrzny czujnik CO2'
   TextField "Text field_8" at 306,346 size 202x23; Text 'Zewnętrzny czujnik CO2'
   TextField "Text field_9" at 569,346 size 206x23; Text 'Stopień zasłonięcia rolet'
   IOField "I/O field_4" at 599,94 size 150x60; FormatPattern 9999
      ProcessValue <- "Czujnik_natezenia_światła"
   IOField "I/O field_5" at 599,242 size 150x60; FormatPattern 999
      ProcessValue <- "Czujnik_wiatru"
   IOField "I/O field_6" at 69,375 size 150x60; FormatPattern 9999
      ProcessValue <- "Wewnetrzny_czujnik_CO2"
   IOField "I/O field_7" at 346,375 size 150x60; FormatPattern 9999
      ProcessValue <- "Zewnetrzny_czujnik_CO2"
   IOField "I/O field_8" at 599,375 size 150x60; FormatPattern 999
      ProcessValue <- "Stopien_zasloniecia_rolet"
   IOField "I/O field_10" at 69,94 size 150x60; FormatPattern 999
      ProcessValue <- "Czujnik_wilgotności_powietrza"
   IOField "I/O field_11" at 346,94 size 150x60; FormatPattern 999
      ProcessValue <- "Czujnik_wilgotności_gleby"
   IOField "I/O field_12" at 69,242 size 150x60; FormatPattern 99.9
      ProcessValue <- "Temperatura_wewnetrzna"
   IOField "I/O field_13" at 346,242 size 150x60; FormatPattern 99.9
      ProcessValue <- "Temperatura_zewnetrzna"
   TextField "Text field_10" at 248,5 size 321x34; Text 'ZAPISZ RECEPTURE / SYMULACJA CZUJNIKÓW'
   Button "Button_1" at 750,0 size 50x50; TextOff 'WRÓĆ'; PictureOff "Back_arrow"
      on Click: function_efd93a16()
   Button "Button_14" at 3,1 size 43x43; TextOff 'DOM'; PictureOff "home_1"
      on Click: ActivateScreen("Root screen", 0)

screen "Root screen" 800x480, template "Template_1"
   on GenerateScreen: SetTag("Tag_ScreenNumber", 0)
   Button "Button_1" at 9,154 size 300x70; TextOff 'TRYB MANUALNY'
      on Click: ActivateScreen("tryb_manualny", 0)
   Button "Button_2" at 10,70 size 300x70; TextOff 'TRYB AUTOMATYCZNY'
      on Click: ActivateScreen("tryb_automatyczny", 0)
   TextField "Text field_2" at 73,1 size 601x52; Text 'AUTOMATYCZNA SZKLARNIA'
   GraphicView "Graphic view_1" at 370,70 size 392x338; Picture "garden-tools-graphic-clipart-design-free-png"
   Button "Button_5" at 10,237 size 300x70; TextOff 'TRYB RECEPTUR'
      on Click: function_e3503463('\USB_X60.1\record.csv', U 0, 2, 1, N); ActivateScreen("Receptury", 0)
   Button "Button_3" at 10,322 size 300x70; TextOff 'SYMULACJA'
      on Click: ActivateScreen("Symulacja_czujnikow", 0)

screen "praca" 800x480
   on GenerateScreen: SetTag("Tag_ScreenNumber", 5); function_ef3f5d25("Alarm window_Unacknowledged", -1)
   GraphicView "Graphic view_4" at 275,402 size 70x70; Picture "soil-sensor_11298794"
   GraphicView "Graphic view_3" at 4,181 size 70x70; Picture "sensor_4212513"
   GraphicView "Graphic view_5" at 268,181 size 70x70; Picture "sensor_4212519"
   GraphicView "Graphic view_1" at 560,402 size 70x70; Picture "fan_4829316"
      Visibility <- "Wentylator"
   GraphicView "Graphic view_6" at 561,276 size 70x70; Picture "heater_4463010"
      Visibility <- "Grzałka"
   GraphicView "Graphic view_7" at 560,170 size 70x70; Picture "irrigation_18631825"
      Visibility <- "Pompa_podlewanie"
   GraphicView "Graphic view_8" at 12,403 size 70x70; Picture "anemometer_1113716"
   GraphicView "Graphic view_9" at 560,402 size 70x70; Picture "fan_off"
      Visibility <- "Wentylator"
   GraphicView "Graphic view_10" at 561,276 size 70x70; Picture "heater_off"
      Visibility <- "Grzałka"
   GraphicView "Graphic view_11" at 560,170 size 70x70; Picture "irrigation_off"
      Visibility <- "Pompa_podlewanie"
   GraphicView "Graphic view_12" at 279,273 size 70x70; Picture "sensor_2828470"
   TextField "Text field_1" at 53,158 size 204x23; Text 'INSOLATION / NASŁONECZNIENIE / SONNENEINSTRAHLUNG'
   TextField "Text field_3" at 45,379 size 166x23; Text 'SZYBKOŚĆ WIATRU'
   TextField "Text field_5" at 290,158 size 223x23; Text 'WILGOTNOŚĆ POWIETRZA'
   TextField "Text field_6" at 319,379 size 175x23; Text 'WILGOTNOŚĆ GLEBY'
   TextField "Text field_7" at 629,154 size 116x23; Text 'PODLEWANIE'
   TextField "Text field_8" at 639,258 size 80x23; Text 'GRZANIE'
   TextField "Text field_9" at 628,379 size 117x23; Text 'WENTYLACJA'
   TextField "Text field_10" at 80,10 size 256x34; Text 'PODGLĄD NA ŻYWO'
   Button "Button_1" at 750,0 size 50x50; TextOff 'WRÓĆ'; PictureOff "Back_arrow"
      on Click: function_efd93a16(); SetBit("HMI_Reset_Trybow")
   Button "Button_2" at 3,1 size 43x43; TextOff 'DOM'; PictureOff "home_1"
      on Click: ActivateScreen("Root screen", 0); SetBit("HMI_Reset_Trybow")
   IOField "I/O field_3" at 95,408 size 70x65; FormatPattern 999
      ProcessValue <- "Czujnik_wiatru"
   IOField "I/O field_5" at 349,283 size 83x65; FormatPattern 9999
      ProcessValue <- "Zewnetrzny_czujnik_CO2"
   IOField "I/O field_4" at 378,178 size 69x65; FormatPattern 999
      ProcessValue <- "Czujnik_wilgotności_powietrza"
   IOField "I/O field_6" at 382,403 size 68x65; FormatPattern 999
      ProcessValue <- "Czujnik_wilgotności_gleby"
   TextField "Text field_12" at 447,196 size 47x46; Text '%'
   TextField "Text field_13" at 467,411 size 47x46; Text '%'
   TextField "Text field_14" at 193,170 size 47x72; Text 'W m²'
   IOField "I/O field_1" at 84,196 size 101x32; FormatPattern 99999
      ProcessValue <- "Czujnik_natezenia_światła"
   TextField "Text field_15" at 174,408 size 52x72; Text 'Km h'
   Circle "Circle_1" at 704,194 size 48x48
      Visibility <- "Pompa_podlewanie"
   Circle "Circle_2" at 703,289 size 48x48
      Visibility <- "Grzałka"
   TextField "Text field_16" at 448,289 size 69x39; Text 'ppm'
   Circle "Circle_4" at 704,194 size 48x48
      Visibility <- "Pompa_podlewanie"
   Circle "Circle_5" at 703,289 size 48x48
      Visibility <- "Grzałka"
   Circle "Circle_3" at 704,421 size 48x48
      Visibility <- "Wentylator"
   Circle "Circle_6" at 704,421 size 48x48
      Visibility <- "Wentylator"
   TextField "Text field_17" at 380,10 size 288x34; Text 'PODGLĄD NA ŻYWO / TRYB AUTOMATYCZNY'
      Visibility <- "HMI_Aktywacja_trybu_automatycznego"
   GraphicView "Graphic view_13" at 561,69 size 70x70; Picture "sprinkler_4552152"
      Visibility <- "Pompa_zraszacze"
   GraphicView "Graphic view_14" at 561,69 size 70x70; Picture "sprinkler"
      Visibility <- "Pompa_zraszacze"
   Circle "Circle_7" at 704,89 size 48x48
      Visibility <- "Pompa_zraszacze"
   Circle "Circle_8" at 704,89 size 48x48
      Visibility <- "Pompa_zraszacze"
   TextField "Text field_19" at 613,58 size 156x23; Text 'PODLEWANIE / MIKROZRASZANIE'
   GraphicView "Graphic view_15" at 1,72 size 70x70; Picture "Thermometer_icon"
   IOField "I/O field_8" at 74,79 size 97x65; FormatPattern 99.99
      ProcessValue <- "Temperatura_wewnetrzna"
   TextField "Text field_21" at 172,91 size 46x46; Text '°C'
   GraphicView "Graphic view_16" at 276,72 size 70x70; Picture "Thermometer_icon"
   IOField "I/O field_9" at 349,79 size 97x65; FormatPattern 99.99
      ProcessValue <- "Temperatura_zewnetrzna"
   TextField "Text field_23" at 448,88 size 46x46; Text '°C'
   TextField "Text field_20" at 59,55 size 137x42; Text 'TEMPERATURA TEMPERATURA WEWNTĘTRZNA'
   TextField "Text field_22" at 336,55 size 132x42; Text 'TEMPERATURA TEMPERATURA ZEWNĘTRZNA'
   GraphicView "Graphic view_2" at 12,279 size 70x70; Picture "sensor_2828470"
   IOField "I/O field_2" at 82,289 size 83x65; FormatPattern 9999
      ProcessValue <- "Wewnetrzny_czujnik_CO2"
   TextField "Text field_11" at 181,295 size 69x39; Text 'ppm'
   TextField "Text field_2" at 84,258 size 124x42; Text 'STĘŻENIE CO2 WEWNĘTRZNE STĘŻENIE CO2'
   TextField "Text field_4" at 353,262 size 123x42; Text 'STĘŻENIE CO2 ZEWNĘTRZNE STĘŻENIE CO2'
   TextField "Text field_18" at 381,10 size 211x34; Text 'TRYB RECEPTUR'
      Visibility <- "HMI_Aktywacja_trybu_Receptur"

screen "Receptury" 800x480
   RecipeView "Recipe view_1" at 0,44 size 799x413; RecipeNameCaption 'Recipe Name: / Wybierz Recepturę / Rezepturname:'; EntryNameCaption 'Entry Name / Zapisane Parametry / Eintragsname'; DataRecordNameCaption 'Data Record Name: / Wybierz Recepturę / Datensatzname:'; Recipe "Receptura_nr1"
   GraphicView "Graphic view_1" at 529,152 size 35x35; Picture "Thermometer_icon"
   GraphicView "Graphic view_2" at 529,190 size 35x35; Picture "sensor_4212519"
   GraphicView "Graphic view_3" at 529,230 size 35x35; Picture "soil-sensor_11298794"
   GraphicView "Graphic view_4" at 529,269 size 35x35; Picture "window_11250237"
   GraphicView "Graphic view_5" at 529,308 size 35x35; Picture "sensor_2828470"
   GraphicView "Graphic view_6" at 529,348 size 35x35; Picture "sensor_4212513"
   TextField "Text field_11" at 569,150 size 39x38; Text '°C'
   TextField "Text field_18" at 569,190 size 39x38; Text '%'
   TextField "Text field_1" at 569,230 size 39x38; Text '%'
   TextField "Text field_2" at 564,269 size 57x32; Text '1/0'
   TextField "Text field_16" at 563,308 size 55x32; Text 'ppm'
   TextField "Text field_6" at 576,339 size 28x50; Text '°C W m'
   TextField "Text field_3" at 593,362 size 31x17; Text '2'
   Button "Button_1" at 750,0 size 50x50; TextOff 'WRÓĆ'; PictureOff "Back_arrow"
      on Click: function_efd93a16()
   Button "Button_14" at 3,1 size 43x43; TextOff 'DOM'; PictureOff "home_1"
      on Click: ActivateScreen("Root screen", 0)
   TextField "Text field_4" at 320,2 size 170x37; Text 'RECEPTURY'
   TextField "Text field_5" at 12,448 size 50x23; Text 'Nowy'
   TextField "Text field_7" at 69,448 size 57x23; Text 'Zapisz'
   TextField "Text field_8" at 137,448 size 45x23; Text 'Usuń'
   TextField "Text field_9" at 197,444 size 47x36; Text 'Zmień Nazwę'
   TextField "Text field_10" at 672,444 size 52x36; Text 'Załaduj z PLC'
   TextField "Text field_12" at 735,444 size 52x36; Text 'Załaduj do PLC'
   Button "Button_2" at 379,406 size 281x40; TextOff 'ZATWIERDŹ'
      on Click: ResetBit("HMI_Reset_Trybow"); ActivateScreen("praca", 0); SetBit("HMI_Aktywacja_trybu_automatycznego")
   TextField "Text field_13" at 435,450 size 173x23; Text 'Przejdź w tryb pracy'
   Button "Button_3" at 282,407 size 50x40; TextOff 'Z'; PictureOff "Graphic_9"
      on Click: function_ea909784(1, U 0, '\USB_X60.1\record.csv', 2, 1, N)
   TextField "Text field_14" at 263,444 size 88x36; Text 'Zapisz Kopię zapasową'

Template "Template_1" 800x480
   Button "Exit" at 671,429 size 71x50; TextOn 'Exit'; TextOff 'Exit'; PictureOn "ExitRuntime_KTP700_Basic_PN_TR"; PictureOff "ExitRuntime_KTP700_Basic_PN_TR"
      on Release: StopRuntime(0)
   Button "Alarms" at 524,429 size 71x50; TextOn 'Alarms'; TextOff 'Alarms'; PictureOn "AlarmDisplay_KTP700_Basic_PN_TR"; PictureOff "AlarmDisplay_KTP700_Basic_PN_TR"
      on Release: function_ef3f5d25("Alarm window_Unacknowledged", -1)
   Button "Start screen" at 169,429 size 71x50; TextOn 'Start screen'; TextOff 'Start screen'; PictureOn "NavigateHome_KTP700_Basic_PN_TR"; PictureOff "NavigateHome_KTP700_Basic_PN_TR"
      on Release: ActivateScreen("Root screen", 0)
      Visibility <- "AlwaysTRUE"
   Button "Language" at 377,429 size 71x50; TextOn 'Language'; TextOff 'Language'; PictureOn "ToggleLanguage_KTP700_Basic_PN_TR"; PictureOff "ToggleLanguage_KTP700_Basic_PN_TR"
      on Release: function_fb9197e8(-1)
*)

(* ===== HMI "HMI_RT_2" =====
system functions are stored by id; their names below are inferred from use
connection "HMI_Connection_3": ETHERNET, SMART_S7_1200_OMS

HMI tags "Default tag table"
   "Tag_ScreenNumber" : Int = PLC HMI.Numer_ekranu_HMI AT %MD0, 100 ms
   "AlwaysTRUE" : Bool = PLC AlwaysTRUE AT %M1.2, 1 s
   "HMI_Aktywacja_trybu_zapis_Receptur" : Bool = PLC HMI.Aktywacja_trybu_zapis_Receptur, 1 s
   "HMI_Aktywacja_trybu_Receptur" : Bool = PLC HMI.Aktywacja_trybu_Receptur, 1 s
   "HMI_Aktywacja_trybu_automatycznego" : Bool = PLC HMI.Aktywacja_trybu_automatycznego, 1 s
   "Tryb_auto_parametry_Temperatura" : Real = PLC Tryb_auto_parametry.Temperatura, 1 s
   "Tryb_auto_parametry_System_okien" : Bool = PLC Tryb_auto_parametry.System_okien, 1 s
   "Tryb_auto_parametry_Wilgotnosc_gleby" : Int = PLC Tryb_auto_parametry.Wilgotnosc_gleby, 1 s
   "Tryb_auto_parametry_Naslonecznienie" : Int = PLC Tryb_auto_parametry.Naslonecznienie, 1 s
   "Tryb_auto_parametry_Stezenie_co2" : Int = PLC Tryb_auto_parametry.Stezenie_co2, 1 s
   "Tryb_auto_parametry_Wilgotnosc_powietrza" : Int = PLC Tryb_auto_parametry.Wilgotnosc_powietrza, 1 s
   "Pompa_zraszacze" : Bool = PLC Pompa_zraszacze AT %Q0.2, 1 s
   "Pompa_podlewanie" : Bool = PLC Pompa_podlewanie AT %Q1.0, 1 s
   "Grzałka" : Bool = PLC Grzałka AT %Q0.0, 1 s
   "Wentylator" : Bool = PLC Wentylator AT %Q0.1, 1 s
   "HMI_Reset_Trybow" : Bool = PLC HMI.Reset_Trybow, 1 s

HMI tags "Do_PLC"
   "System_okien_auto" : Bool = PLC HMI.System_okien_auto, 500 ms
   "Stopien_zasloniecia_rolet_manual" : Int = PLC HMI.Stopien_zasloniecia_rolet_manual, 100 ms
   "Przycisk_zraszania_manual" : Bool = PLC HMI.Przycisk_zraszacze_manual AT %Q0.2, 100 ms
   "Przycisk_wentylacja_manual" : Bool = PLC HMI.Przycisk_wentylacja_manual AT %Q0.1, 100 ms
   "Przycisk_grzanie_manual" : Bool = PLC HMI.Przycisk_grzanie_manual AT %Q0.0, 100 ms
   "Otwarcie_okien_man" : Bool = PLC HMI.Otwarcie_okien_manual AT %DB1.DBW0, 100 ms
   "Temperatura_auto" : Real = PLC HMI.Temperatura_auto, 500 ms
   "Naslonecznienie_auto" : Int = PLC HMI.Naslonecznienie_auto AT %DB1.DBW0, 500 ms
   "Wilgotnosc_powietrza_auto" : Int = PLC HMI.Wilgotnosc_powietrza_auto AT %DB1.DBW0, 500 ms
   "Wilgotnosc_gleby_auto" : Int = PLC HMI.Wilgotnosc_gleby_auto AT %DB1.DBW0, 500 ms
   "Przycisk_zatwierdz_auto" : Bool = PLC HMI.Przycisk_zatwierdz_auto AT %DB1.DBW0, 100 ms
   "nazwa_receptury" : String[254] = PLC HMI.nazwa_receptury AT %DB1.DBX0.0, 500 ms
   "przycisk_zatwierdz_zapis_receptury" : Bool = PLC HMI.Przycisk_zatwierdz_zapis_receptury AT %DB1.DBX0.0, 500 ms
   "HMI_Przycisk_zatwierdz_wybor_receptury" : Bool = PLC HMI.Przycisk_zatwierdz_wybor_receptury AT %DB1.DBX0.0, 500 ms
   "Przycisk_podlewania_manual" : Bool = PLC HMI.Przycisk_podlewanie_manual AT %Q0.2, 100 ms
   "Poziom_CO2_auto" : Int = PLC HMI.Poziom_CO2_auto AT %DB1.DBX0.0, 1 s

HMI tags "Z_PLC"
   "Czujnik_wilgotności_powietrza" : Int = PLC Wejscia_PLC.Czujnik_wilgotności_powietrza, 500 ms
   "Temperatura_wewnetrzna" : Real = PLC Wejscia_PLC.Temperatura_wewnetrzna, 500 ms
   "Czujnik_natezenia_światła" : Int = PLC Wejscia_PLC.Czujnik_natezenia_swiatła, 500 ms
   "Czujnik_wilgotności_gleby" : Int = PLC Wejscia_PLC.Czujnik_wilgotności_gleby, 500 ms
   "Wewnetrzny_czujnik_CO2" : Int = PLC Wejscia_PLC.Wewnetrzny_czujnik_CO2, 500 ms
   "Czujnik_wiatru" : Int = PLC Wejscia_PLC.Czujnik_wiatru, 500 ms
   "Stopien_zasloniecia_rolet" : Int = PLC Wejscia_PLC.Stopien_zasloniecia_rolet, 1 s
   "Zewnetrzny_czujnik_CO2" : Int = PLC Wejscia_PLC.Zewnetrzny_czujnik_CO2 AT %DB1.DBW0, 1 s
   "Temperatura_zewnetrzna" : Real = PLC Wejscia_PLC.Temperatura_zewnetrzna AT %DB1.DBW0, 1 s

analog alarms
   1: 'Stężenie CO2 ma powyżej 3000 jednostek / Stężenie CO2 ma powyżej 3000 jednostek, dłużesze przebywanie w takim środowisku może być szkodliwe dla człowieka. Zalecane jest włączenie wentylacji lub otworzenie okien.', class Warnings, trigger "Wewnetrzny_czujnik_CO2"
   2: 'Temperatura powyżej 35 stopni / Temperatura powyżej 35 stopni, zaleca się wyłączenie grzania.', class Warnings, trigger "Temperatura_wewnetrzna"
   3: 'Podmuchy wiatru osiągają wartości powyżej 35 km/h, system automatyczny zamyka okna.', class Warnings, trigger "Czujnik_wiatru"
   4: 'Stężenie CO2 ma powyżej 5000 jednostek. NIEZWŁOCZNIE OTWORZ OKNA ORAZ ZAŁĄCZ WENTYLATOR, NASTĘPNIE NALEŻY EWAKUOWAĆ WSZYSTKUCH ZNAJDUJĄCYCH SIĘ W POMIESZCZENIU / Stężenie CO2 ma powyżej 5000 jednostek. NIEZWŁOCZNIE OTWORZ OKNA ORAZ ZAŁĄCZ WENTYLATOR, NASTĘPNIE NALEŻY EWAKUOWAĆ WSZYSTKUCH ZNAJDUJĄCYCH SIĘ W POMIESZCZENIU', class Errors, trigger "Wewnetrzny_czujnik_CO2"
   5: 'Temperatura powyżej 45 stopni, NIEZWŁOCZNIE SPRAWDŹ DZIAŁANIE GRZAŁKI, TERMOMETRU LUB WENTYLATORA. / Temperatura powyżej 45 stopni, NIEZWŁOCZNIE SPRAWDŹ DZIAŁANIE GRZAŁKI, TERMOMETRU LUB WENTYLATORA. JEŚLI TEMPERATURA NIE SPADA ZALECA SIĘ EWAKUOWAĆ WSZYSTKICH PRZEBYWAJĄCYCH W POMIESZCZENIU', class Errors, trigger "Temperatura_wewnetrzna"

text list "receptury": 0..1 ''

recipe "Receptura_nr1": Temperatura <- "Tryb_auto_parametry_Temperatura", Wilgotność Powietrza <- "Tryb_auto_parametry_Wilgotnosc_powietrza", Wilgotność gleby <- "Tryb_auto_parametry_Wilgotnosc_gleby", System okien <- "Tryb_auto_parametry_System_okien", Stężenie CO2 <- "Tryb_auto_parametry_Stezenie_co2", Nasłonecznienie <- "Tryb_auto_parametry_Naslonecznienie"

screen "Root screen" 800x480, template "Template_1"
   on GenerateScreen: SetTag("Tag_ScreenNumber", 0)
   Button "Button_1" at 9,154 size 300x70; TextOff 'TRYB MANUALNY'
      on Click: ActivateScreen("tryb_manualny", 0)
   Button "Button_2" at 10,70 size 300x70; TextOff 'TRYB AUTOMATYCZNY'
      on Click: ActivateScreen("tryb_automatyczny", 0)
   TextField "Text field_2" at 73,1 size 601x52; Text 'AUTOMATYCZNA SZKLARNIA'
   GraphicView "Graphic view_1" at 370,70 size 392x338; Picture "garden-tools-graphic-clipart-design-free-png"
   Button "Button_5" at 10,237 size 300x70; TextOff 'TRYB RECEPTUR'
      on Click: function_e3503463('\USB_X60.1\record.csv', U 0, 2, 1, N); ActivateScreen("Receptury", 0)
   Button "Button_3" at 10,322 size 300x70; TextOff 'SYMULACJA'
      on Click: ActivateScreen("Symulacja_czujnikow", 0)

screen "tryb_manualny" 800x480
   on GenerateScreen: SetTag("Tag_ScreenNumber", 2)
   TextField "Text field_1" at 295,7 size 223x34; Text 'TRYB MANUALNY'
   TextField "Text field_4" at 512,155 size 171x61; Text 'STOPIEŃ OTWARCIA OKIEN OTWIERANIE OKIEN'
   Button "Button_4" at 518,261 size 80x70; TextOff 'PODLEWANIE'
      on Click: InvertBit("Przycisk_podlewania_manual")
   Button "Button_5" at 611,261 size 80x70; TextOff 'GRZANIE'
      on Click: InvertBit("Przycisk_grzanie_manual")
   Button "Button_6" at 701,261 size 80x70; TextOff 'WENTYLACJA'
      on Click: InvertBit("Przycisk_wentylacja_manual")
   GraphicView "Graphic view_1" at 710,356 size 60x60; Picture "fan_4829316"
      Visibility <- "Wentylator"
   GraphicView "Graphic view_6" at 622,356 size 60x60; Picture "heater_4463010"
      Visibility <- "Grzałka"
   GraphicView "Graphic view_7" at 527,356 size 64x60; Picture "irrigation_18631825"
      Visibility <- "Pompa_podlewanie"
   GraphicView "Graphic view_9" at 710,356 size 60x60; Picture "fan_off"
      Visibility <- "Wentylator"
   GraphicView "Graphic view_10" at 622,356 size 60x60; Picture "heater_off"
      Visibility <- "Grzałka"
   GraphicView "Graphic view_11" at 527,356 size 64x60; Picture "irrigation_off"
      Visibility <- "Pompa_podlewanie"
   Button "Button_14" at 6,7 size 43x43; TextOff 'DOM'; PictureOff "home_1"
      on Click: ActivateScreen("Root screen", 0)
   Button "Button_1" at 740,0 size 60x60; TextOff 'Text'; PictureOff "Back_arrow"
      on Click: function_efd93a16()
   Circle "Circle_1" at 541,428 size 42x42
      Visibility <- "Pompa_podlewanie"
   Circle "Circle_4" at 541,428 size 42x42
      Visibility <- "Pompa_podlewanie"
   Circle "Circle_2" at 631,428 size 42x42
      Visibility <- "Grzałka"
   Circle "Circle_5" at 631,428 size 42x42
      Visibility <- "Grzałka"
   Circle "Circle_3" at 720,428 size 41x41
      Visibility <- "Wentylator"
   Circle "Circle_6" at 720,428 size 41x41
      Visibility <- "Wentylator"
   TextField "Text field_8" at 405,71 size 117x61; Text 'STOPIEŃ OTWARCIA OKIEN STOPIEŃ ZASŁONIECIA ROLET'
   Bar "Bar_6" at 624,82 size 165x66; MinimumValue 0; MaximumValue 100
      ProcessValue <- "Stopien_zasloniecia_rolet_manual"
   Button "Button_3" at 530,114 size 80x50; TextOff '+ / ODSŁOŃ'
      on Click: function_b9b71300("Stopien_zasloniecia_rolet_manual", 5)
   Button "Button_7" at 530,60 size 80x50; TextOff '- / ZASŁOŃ'
      on Press: function_dd21b452("Stopien_zasloniecia_rolet_manual", 5)
   Button "Button_2" at 425,261 size 80x70; TextOff 'PODLEWANIE / MIKROZRASZANIE'
      on Click: InvertBit("Przycisk_zraszania_manual")
   GraphicView "Graphic view_2" at 434,356 size 60x60; Picture "sprinkler_4552152"
      Visibility <- "Pompa_zraszacze"
   GraphicView "Graphic view_3" at 434,356 size 60x60; Picture "sprinkler"
      Visibility <- "Pompa_zraszacze"
   Circle "Circle_7" at 443,428 size 42x42
      Visibility <- "Pompa_zraszacze"
   Circle "Circle_8" at 443,428 size 42x42
      Visibility <- "Pompa_zraszacze"
   Switch "Switch_1" at 499,199 size 209x37; CaptionText 'Switch'; TextOff 'ZAMKNIĘTE'; TextOn 'OTWARTE'
      ProcessValue <- "Otwarcie_okien_man"
   TextField "Text field_3" at 11,375 size 166x23; Text 'SZYBKOŚĆ WIATRU'
   IOField "I/O field_3" at 62,407 size 70x65; FormatPattern 999
      ProcessValue <- "Czujnik_wiatru"
   IOField "I/O field_1" at 48,189 size 101x32; FormatPattern 99999
      ProcessValue <- "Czujnik_natezenia_światła"
   TextField "Text field_15" at 129,408 size 52x72; Text 'Km h'
   IOField "I/O field_2" at 44,292 size 83x65; FormatPattern 9999
      ProcessValue <- "Wewnetrzny_czujnik_CO2"
   TextField "Text field_11" at 118,301 size 69x39; Text 'ppm'
   TextField "Text field_5" at 14,148 size 204x23; Text 'INSOLATION / NASŁONECZNIENIE / SONNENEINSTRAHLUNG'
   IOField "I/O field_8" at 58,95 size 93x40; FormatPattern 99.99
      ProcessValue <- "Temperatura_wewnetrzna"
   TextField "Text field_20" at 30,56 size 137x42; Text 'TEMPERATURA TEMPERATURA WEWNTĘTRZNA'
   TextField "Text field_7" at 200,375 size 175x23; Text 'WILGOTNOŚĆ GLEBY'
   IOField "I/O field_5" at 248,293 size 83x65; FormatPattern 9999
      ProcessValue <- "Zewnetrzny_czujnik_CO2"
   IOField "I/O field_4" at 266,174 size 69x65; FormatPattern 999
      ProcessValue <- "Czujnik_wilgotności_powietrza"
   IOField "I/O field_6" at 261,405 size 68x65; FormatPattern 999
      ProcessValue <- "Czujnik_wilgotności_gleby"
   TextField "Text field_12" at 324,182 size 47x46; Text '%'
   TextField "Text field_13" at 321,416 size 47x46; Text '%'
   TextField "Text field_16" at 326,292 size 69x39; Text 'ppm'
   IOField "I/O field_9" at 248,85 size 97x65; FormatPattern 99.99
      ProcessValue <- "Temperatura_zewnetrzna"
   TextField "Text field_23" at 333,90 size 46x46; Text '°C'
   TextField "Text field_22" at 229,57 size 132x42; Text 'TEMPERATURA TEMPERATURA ZEWNĘTRZNA'
   TextField "Text field_9" at 229,256 size 123x42; Text 'STĘŻENIE CO2 ZEWNĘTRZNE STĘŻENIE CO2'
   TextField "Text field_6" at 180,143 size 223x42; Text 'WILGOTNOŚĆ POWIETRZA WILGOTNOŚĆ POWIETRZA'
   TextField "Text field_14" at 140,170 size 47x72; Text 'W m²'
   TextField "Text field_21" at 141,90 size 46x46; Text '°C'
   GraphicView "Graphic view_4" at 419,176 size 60x60; Picture "window_11250237"
   GraphicView "Graphic view_5" at 197,182 size 50x50; Picture "sensor_4212519"
   GraphicView "Graphic view_8" at 4,182 size 50x50; Picture "sensor_4212513"
   GraphicView "Graphic view_12" at 3,87 size 50x50; Picture "Thermometer_icon"
   GraphicView "Graphic view_13" at 199,87 size 50x50; Picture "Thermometer_icon"
   GraphicView "Graphic view_14" at 3,302 size 40x40; Picture "sensor_2828470"
   GraphicView "Graphic view_15" at 197,300 size 40x40; Picture "sensor_2828470"
   GraphicView "Graphic view_16" at 198,412 size 50x50; Picture "soil-sensor_11298794"
   GraphicView "Graphic view_17" at 3,416 size 50x50; Picture "anemometer_1113716"
   TextField "Text field_2" at 27,256 size 124x42; Text 'STĘŻENIE CO2 WEWNĘTRZNE STĘŻENIE CO2'

screen "praca" 800x480
   on GenerateScreen: SetTag("Tag_ScreenNumber", 5); function_ef3f5d25("Alarm window_Unacknowledged", -1)
   GraphicView "Graphic view_4" at 275,402 size 70x70; Picture "soil-sensor_11298794"
   GraphicView "Graphic view_3" at 4,181 size 70x70; Picture "sensor_4212513"
   GraphicView "Graphic view_5" at 268,181 size 70x70; Picture "sensor_4212519"
   GraphicView "Graphic view_1" at 560,402 size 70x70; Picture "fan_4829316"
      Visibility <- "Wentylator"
   GraphicView "Graphic view_6" at 561,276 size 70x70; Picture "heater_4463010"
      Visibility <- "Grzałka"
   GraphicView "Graphic view_7" at 560,170 size 70x70; Picture "irrigation_18631825"
      Visibility <- "Pompa_podlewanie"
   GraphicView "Graphic view_8" at 12,403 size 70x70; Picture "anemometer_1113716"
   GraphicView "Graphic view_9" at 560,402 size 70x70; Picture "fan_off"
      Visibility <- "Wentylator"
   GraphicView "Graphic view_10" at 561,276 size 70x70; Picture "heater_off"
      Visibility <- "Grzałka"
   GraphicView "Graphic view_11" at 560,170 size 70x70; Picture "irrigation_off"
      Visibility <- "Pompa_podlewanie"
   GraphicView "Graphic view_12" at 279,273 size 70x70; Picture "sensor_2828470"
   TextField "Text field_1" at 53,158 size 204x23; Text 'INSOLATION / NASŁONECZNIENIE / SONNENEINSTRAHLUNG'
   TextField "Text field_3" at 45,379 size 166x23; Text 'SZYBKOŚĆ WIATRU'
   TextField "Text field_5" at 290,158 size 223x23; Text 'WILGOTNOŚĆ POWIETRZA'
   TextField "Text field_6" at 319,379 size 175x23; Text 'WILGOTNOŚĆ GLEBY'
   TextField "Text field_7" at 629,154 size 116x23; Text 'PODLEWANIE'
   TextField "Text field_8" at 639,258 size 80x23; Text 'GRZANIE'
   TextField "Text field_9" at 628,379 size 117x23; Text 'WENTYLACJA'
   TextField "Text field_10" at 80,10 size 256x34; Text 'PODGLĄD NA ŻYWO'
   Button "Button_1" at 750,0 size 50x50; TextOff 'WRÓĆ'; PictureOff "Back_arrow"
      on Click: function_efd93a16(); SetBit("HMI_Reset_Trybow")
   Button "Button_2" at 3,1 size 43x43; TextOff 'DOM'; PictureOff "home_1"
      on Click: ActivateScreen("Root screen", 0); SetBit("HMI_Reset_Trybow")
   IOField "I/O field_3" at 95,408 size 70x65; FormatPattern 999
      ProcessValue <- "Czujnik_wiatru"
   IOField "I/O field_5" at 349,283 size 83x65; FormatPattern 9999
      ProcessValue <- "Zewnetrzny_czujnik_CO2"
   IOField "I/O field_4" at 378,178 size 69x65; FormatPattern 999
      ProcessValue <- "Czujnik_wilgotności_powietrza"
   IOField "I/O field_6" at 382,403 size 68x65; FormatPattern 999
      ProcessValue <- "Czujnik_wilgotności_gleby"
   TextField "Text field_12" at 447,196 size 47x46; Text '%'
   TextField "Text field_13" at 467,411 size 47x46; Text '%'
   TextField "Text field_14" at 193,170 size 47x72; Text 'W m²'
   IOField "I/O field_1" at 84,196 size 101x32; FormatPattern 99999
      ProcessValue <- "Czujnik_natezenia_światła"
   TextField "Text field_15" at 174,408 size 52x72; Text 'Km h'
   Circle "Circle_1" at 704,194 size 48x48
      Visibility <- "Pompa_podlewanie"
   Circle "Circle_2" at 703,289 size 48x48
      Visibility <- "Grzałka"
   TextField "Text field_16" at 448,289 size 69x39; Text 'ppm'
   Circle "Circle_4" at 704,194 size 48x48
      Visibility <- "Pompa_podlewanie"
   Circle "Circle_5" at 703,289 size 48x48
      Visibility <- "Grzałka"
   Circle "Circle_3" at 704,421 size 48x48
      Visibility <- "Wentylator"
   Circle "Circle_6" at 704,421 size 48x48
      Visibility <- "Wentylator"
   TextField "Text field_17" at 380,10 size 288x34; Text 'PODGLĄD NA ŻYWO / TRYB AUTOMATYCZNY'
      Visibility <- "HMI_Aktywacja_trybu_automatycznego"
   GraphicView "Graphic view_13" at 561,69 size 70x70; Picture "sprinkler_4552152"
      Visibility <- "Pompa_zraszacze"
   GraphicView "Graphic view_14" at 561,69 size 70x70; Picture "sprinkler"
      Visibility <- "Pompa_zraszacze"
   Circle "Circle_7" at 704,89 size 48x48
      Visibility <- "Pompa_zraszacze"
   Circle "Circle_8" at 704,89 size 48x48
      Visibility <- "Pompa_zraszacze"
   TextField "Text field_19" at 613,58 size 156x23; Text 'PODLEWANIE / MIKROZRASZANIE'
   GraphicView "Graphic view_15" at 1,72 size 70x70; Picture "Thermometer_icon"
   IOField "I/O field_8" at 74,79 size 97x65; FormatPattern 99.99
      ProcessValue <- "Temperatura_wewnetrzna"
   TextField "Text field_21" at 172,91 size 46x46; Text '°C'
   GraphicView "Graphic view_16" at 276,72 size 70x70; Picture "Thermometer_icon"
   IOField "I/O field_9" at 349,79 size 97x65; FormatPattern 99.99
      ProcessValue <- "Temperatura_zewnetrzna"
   TextField "Text field_23" at 448,88 size 46x46; Text '°C'
   TextField "Text field_20" at 59,55 size 137x42; Text 'TEMPERATURA TEMPERATURA WEWNTĘTRZNA'
   TextField "Text field_22" at 336,55 size 132x42; Text 'TEMPERATURA TEMPERATURA ZEWNĘTRZNA'
   GraphicView "Graphic view_2" at 12,279 size 70x70; Picture "sensor_2828470"
   IOField "I/O field_2" at 82,289 size 83x65; FormatPattern 9999
      ProcessValue <- "Wewnetrzny_czujnik_CO2"
   TextField "Text field_11" at 181,295 size 69x39; Text 'ppm'
   TextField "Text field_2" at 84,258 size 124x42; Text 'STĘŻENIE CO2 WEWNĘTRZNE STĘŻENIE CO2'
   TextField "Text field_4" at 353,262 size 123x42; Text 'STĘŻENIE CO2 ZEWNĘTRZNE STĘŻENIE CO2'
   TextField "Text field_18" at 381,10 size 211x34; Text 'TRYB RECEPTUR'
      Visibility <- "HMI_Aktywacja_trybu_Receptur"

Template "Template_1" 800x480
   Button "Exit" at 671,429 size 71x50; TextOn 'Exit'; TextOff 'Exit'; PictureOn "ExitRuntime_KTP700_Basic_PN_TR"; PictureOff "ExitRuntime_KTP700_Basic_PN_TR"
      on Release: StopRuntime(0)
   Button "Alarms" at 524,429 size 71x50; TextOn 'Alarms'; TextOff 'Alarms'; PictureOn "AlarmDisplay_KTP700_Basic_PN_TR"; PictureOff "AlarmDisplay_KTP700_Basic_PN_TR"
      on Release: function_ef3f5d25("Alarm window_Unacknowledged", -1)
   Button "Start screen" at 169,429 size 71x50; TextOn 'Start screen'; TextOff 'Start screen'; PictureOn "NavigateHome_KTP700_Basic_PN_TR"; PictureOff "NavigateHome_KTP700_Basic_PN_TR"
      on Release: ActivateScreen("Root screen", 0)
      Visibility <- "AlwaysTRUE"
   Button "Language" at 377,429 size 71x50; TextOn 'Language'; TextOff 'Language'; PictureOn "ToggleLanguage_KTP700_Basic_PN_TR"; PictureOff "ToggleLanguage_KTP700_Basic_PN_TR"
      on Release: function_fb9197e8(-1)

screen "Receptury" 800x480
   RecipeView "Recipe view_1" at 0,44 size 799x413; Recipe "Receptura_nr1"; RecipeNameCaption 'Recipe Name: / Wybierz Recepturę / Rezepturname:'; EntryNameCaption 'Entry Name / Zapisane Parametry / Eintragsname'; DataRecordNameCaption 'Data Record Name: / Wybierz Recepturę / Datensatzname:'
   GraphicView "Graphic view_1" at 529,152 size 35x35; Picture "Thermometer_icon"
   GraphicView "Graphic view_2" at 529,190 size 35x35; Picture "sensor_4212519"
   GraphicView "Graphic view_3" at 529,230 size 35x35; Picture "soil-sensor_11298794"
   GraphicView "Graphic view_4" at 529,269 size 35x35; Picture "window_11250237"
   GraphicView "Graphic view_5" at 529,308 size 35x35; Picture "sensor_2828470"
   GraphicView "Graphic view_6" at 529,348 size 35x35; Picture "sensor_4212513"
   TextField "Text field_11" at 569,150 size 39x38; Text '°C'
   TextField "Text field_18" at 569,190 size 39x38; Text '%'
   TextField "Text field_1" at 569,230 size 39x38; Text '%'
   TextField "Text field_2" at 564,269 size 57x32; Text '1/0'
   TextField "Text field_16" at 563,308 size 55x32; Text 'ppm'
   TextField "Text field_6" at 576,339 size 28x50; Text '°C W m'
   TextField "Text field_3" at 593,362 size 31x17; Text '2'
   Button "Button_1" at 750,0 size 50x50; TextOff 'WRÓĆ'; PictureOff "Back_arrow"
      on Click: function_efd93a16()
   Button "Button_14" at 3,1 size 43x43; TextOff 'DOM'; PictureOff "home_1"
      on Click: ActivateScreen("Root screen", 0)
   TextField "Text field_4" at 320,2 size 170x37; Text 'RECEPTURY'
   TextField "Text field_5" at 12,448 size 50x23; Text 'Nowy'
   TextField "Text field_7" at 69,448 size 57x23; Text 'Zapisz'
   TextField "Text field_8" at 137,448 size 45x23; Text 'Usuń'
   TextField "Text field_9" at 197,444 size 47x36; Text 'Zmień Nazwę'
   TextField "Text field_10" at 672,444 size 52x36; Text 'Załaduj z PLC'
   TextField "Text field_12" at 735,444 size 52x36; Text 'Załaduj do PLC'
   Button "Button_2" at 379,406 size 281x40; TextOff 'ZATWIERDŹ'
      on Click: ResetBit("HMI_Reset_Trybow"); ActivateScreen("praca", 0); SetBit("HMI_Aktywacja_trybu_Receptur")
   TextField "Text field_13" at 435,450 size 173x23; Text 'Przejdź w tryb pracy'
   Button "Button_3" at 282,407 size 50x40; TextOff 'Z'; PictureOff "Graphic_9"
      on Click: function_ea909784(1, U 0, '\USB_X60.1\record.csv', 2, 1, N)
   TextField "Text field_14" at 263,444 size 88x36; Text 'Zapisz Kopię zapasową'

